// TIA Portal V16 export
// export: Created 2022-02-11T14:53:34.4841249Z, ExportSetting WithDefaults, DisplayName Totally Integrated Automation Portal, DisplayVersion V16 Update 1, DisplayName TIA Portal Version Control Interface, DisplayVersion V16, DisplayName TIA Portal Openness, DisplayVersion V16, DisplayName SINAMICS Startdrive Advanced, DisplayVersion V16 Update 5, DisplayName SINAMICS Startdrive G130, G150, S120, S150, SINAMICS MV, S210, DisplayVersion V16 Update 5, DisplayName SINAMICS Startdrive G110M, G120, G120C, G120D, G120P, G115D, DisplayVersion V16 Update 5, DisplayName STEP 7 Professional, DisplayVersion V16, DisplayName STEP 7 Safety, DisplayVersion V16, DisplayName WinCC Advanced, DisplayVersion V16, DisplayName SIMATIC Visualization Architect, DisplayVersion V16
FUNCTION_BLOCK "Сортировка"   // FB9, LAD
VERSION : 0.1
// Логика работы ПФМ
// stored: AutoNumber true, IsIECCheckEnabled false, UDAEnableTagReadback false
   VAR_INPUT
      packet_released : Bool;
   END_VAR
   VAR DB_SPECIFIC
      "TrigE76.4" : Bool;
      Trig_Dovod : Bool;
      LiftPushingPacket : Bool;
      TrigAutoPFM : Bool;
      Trig_Vill : Bool;
      Trig_Vill2 : Bool;
      LiftDownTrig : Bool;
      HaveSxema : Bool;
      NewPacket : Bool;
      LiftDown_old : Bool;
      LiftPushing_old : Bool;
      ForksForcingFinish : Bool;
      LiftForcingFinish : Bool;
      CommonForcingPacket : Bool;
      ElevatorLowering : Bool;
      NoGasketMode : Bool;   // режим без прокладки
      RampIsOn : Bool;
      RampIsOff : Bool;
      power_Vill : Bool := true;
      MakedLayer : Bool;
      AlarmLowerElevator : Bool;
      AlarmNotReadedPack : Bool;
      lift_return_trig : Bool;
      ramp_sync_old : Bool;
      BoardInLayerCounter : Int;
      LayersCounter : Int;
   END_VAR
   VAR
      Vibrator_KeyFazer { S7_SetPoint := 'True'} : "Vibrator";
      Run323_timer { S7_SetPoint := 'True'} : TP;
      LayerCounter { S7_SetPoint := 'True'} : "Adder";
   END_VAR
   VAR_TEMP
      Sert : Word;
   END_VAR
   VAR_TEMP   // added for the SCL form of the ladder/FBD networks
      _w1 : Bool;
      _w2 : Bool;
      _s5time1 : S5Time;
      _w3 : Bool;
      _w4 : Bool;
      _w5 : Bool;
      _s5time2 : S5Time;
   END_VAR
BEGIN

REGION Network 1: 221 группа на 14 моторов общий сигнал готовности
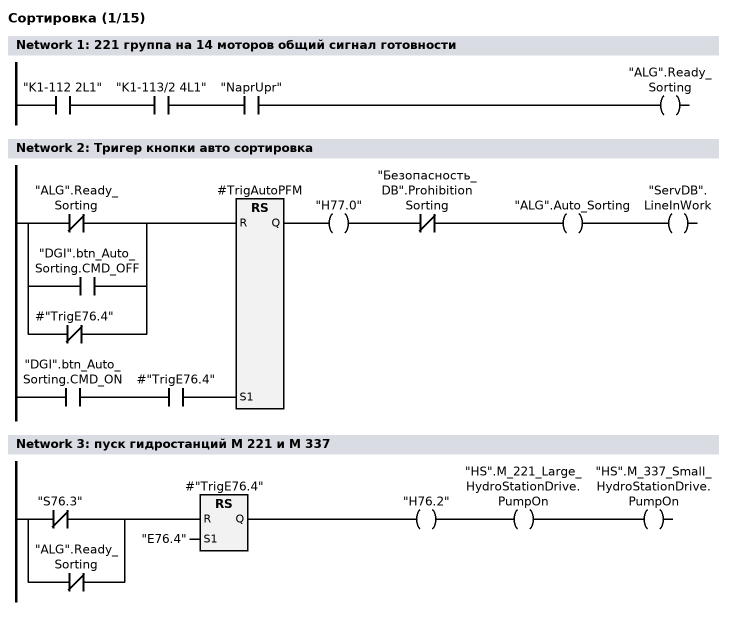
   RUNG wire#powerrail
      Contact( "K1-112 2L1" )
      Contact( "K1-113/2 4L1" )
      Contact( "NaprUpr" )
      Coil( "ALG".Ready_Sorting )
   END_RUNG
   // the same network as SCL:
   "ALG".Ready_Sorting := "K1-112 2L1" AND "K1-113/2 4L1" AND "NaprUpr";
END_REGION

REGION Network 2: Тригер кнопки авто сортировка
   RUNG wire#powerrail
      I_Contact( "ALG".Ready_Sorting )
      wire#w1
      S_RS(operand := #TrigAutoPFM, s1 := wire#w2)
      Coil( "H77.0" )
      I_Contact( "Безопасность_DB".ProhibitionSorting )
      Coil( "ALG".Auto_Sorting )
      Coil( "ServDB".LineInWork )
   END_RUNG
   RUNG wire#powerrail
      Contact( "DGI".btn_Auto_Sorting.CMD_OFF )
   END_RUNG wire#w1
   RUNG wire#powerrail
      I_Contact( #"TrigE76.4" )
   END_RUNG wire#w1
   RUNG wire#powerrail
      Contact( "DGI".btn_Auto_Sorting.CMD_ON )
      Contact( #"TrigE76.4" )
   END_RUNG wire#w2
   // the same network as SCL:
   IF NOT "ALG".Ready_Sorting OR "DGI".btn_Auto_Sorting.CMD_OFF OR NOT #"TrigE76.4" THEN
       #TrigAutoPFM := FALSE;   // RS flip-flop
   END_IF;
   IF "DGI".btn_Auto_Sorting.CMD_ON AND #"TrigE76.4" THEN #TrigAutoPFM := TRUE; END_IF;
   "H77.0" := #TrigAutoPFM;
   "ALG".Auto_Sorting := #TrigAutoPFM AND NOT "Безопасность_DB".ProhibitionSorting;
   "ServDB".LineInWork := "ALG".Auto_Sorting;
END_REGION

REGION Network 3: пуск гидростанций М 221 и M 337
   RUNG wire#powerrail
      I_Contact( "S76.3" )
      wire#w1
      S_RS(operand := #"TrigE76.4", s1 := "E76.4")
      Coil( "H76.2" )
      Coil( "HS".M_221_Large_HydroStationDrive.PumpOn )
      Coil( "HS".M_337_Small_HydroStationDrive.PumpOn )
   END_RUNG
   RUNG wire#powerrail
      I_Contact( "ALG".Ready_Sorting )
   END_RUNG wire#w1
   // the same network as SCL:
   IF NOT "S76.3" OR NOT "ALG".Ready_Sorting THEN
       #"TrigE76.4" := FALSE;   // RS flip-flop
   END_IF;
   IF "E76.4" THEN #"TrigE76.4" := TRUE; END_IF;
   "H76.2" := #"TrigE76.4";
   "HS".M_221_Large_HydroStationDrive.PumpOn := #"TrigE76.4";
   "HS".M_337_Small_HydroStationDrive.PumpOn := #"TrigE76.4";
END_REGION

REGION Network 4: Генерация аварии
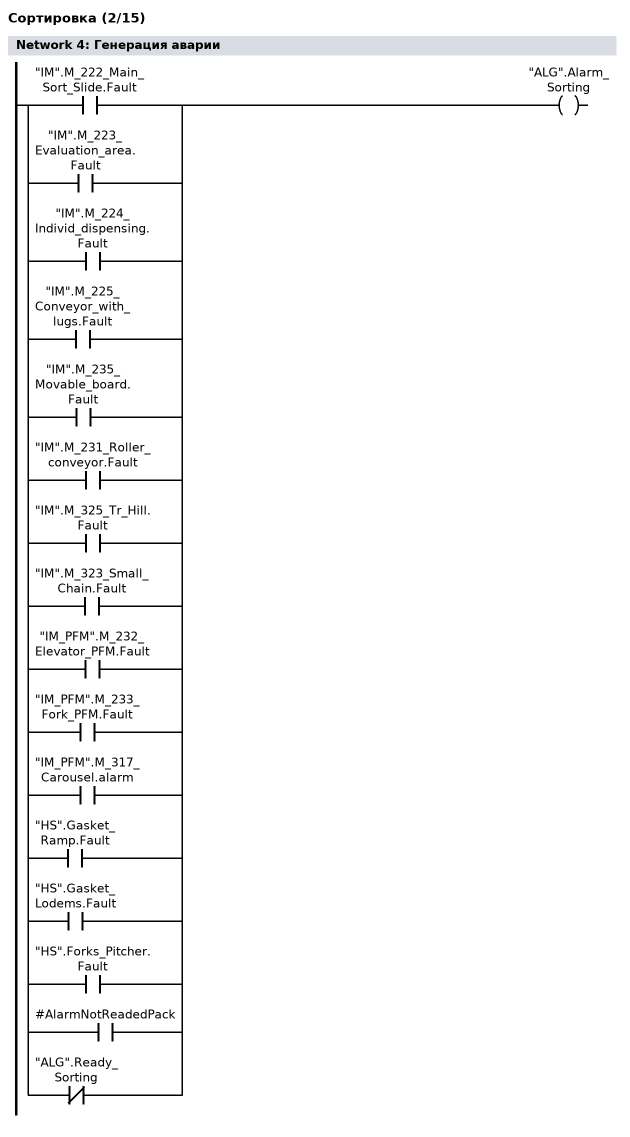
   RUNG wire#powerrail
      Contact( "IM".M_222_Main_Sort_Slide.Fault )
      wire#w1
      Coil( "ALG".Alarm_Sorting )
   END_RUNG
   RUNG wire#powerrail
      Contact( "IM".M_223_Evaluation_area.Fault )
   END_RUNG wire#w1
   RUNG wire#powerrail
      Contact( "IM".M_224_Individ_dispensing.Fault )
   END_RUNG wire#w1
   RUNG wire#powerrail
      Contact( "IM".M_225_Conveyor_with_lugs.Fault )
   END_RUNG wire#w1
   RUNG wire#powerrail
      Contact( "IM".M_235_Movable_board.Fault )
   END_RUNG wire#w1
   RUNG wire#powerrail
      Contact( "IM".M_231_Roller_conveyor.Fault )
   END_RUNG wire#w1
   RUNG wire#powerrail
      Contact( "IM".M_325_Tr_Hill.Fault )
   END_RUNG wire#w1
   RUNG wire#powerrail
      Contact( "IM".M_323_Small_Chain.Fault )
   END_RUNG wire#w1
   RUNG wire#powerrail
      Contact( "IM_PFM".M_232_Elevator_PFM.Fault )
   END_RUNG wire#w1
   RUNG wire#powerrail
      Contact( "IM_PFM".M_233_Fork_PFM.Fault )
   END_RUNG wire#w1
   RUNG wire#powerrail
      Contact( "IM_PFM".M_317_Carousel.alarm )
   END_RUNG wire#w1
   RUNG wire#powerrail
      Contact( "HS".Gasket_Ramp.Fault )
   END_RUNG wire#w1
   RUNG wire#powerrail
      Contact( "HS".Gasket_Lodems.Fault )
   END_RUNG wire#w1
   RUNG wire#powerrail
      Contact( "HS".Forks_Pitcher.Fault )
   END_RUNG wire#w1
   RUNG wire#powerrail
      Contact( #AlarmNotReadedPack )
   END_RUNG wire#w1
   RUNG wire#powerrail
      I_Contact( "ALG".Ready_Sorting )
   END_RUNG wire#w1
   // the same network as SCL:
   "ALG".Alarm_Sorting := "IM".M_222_Main_Sort_Slide.Fault OR "IM".M_223_Evaluation_area.Fault OR "IM".M_224_Individ_dispensing.Fault OR "IM".M_225_Conveyor_with_lugs.Fault OR "IM".M_235_Movable_board.Fault OR "IM".M_231_Roller_conveyor.Fault OR "IM".M_325_Tr_Hill.Fault OR "IM".M_323_Small_Chain.Fault OR "IM_PFM".M_232_Elevator_PFM.Fault OR "IM_PFM".M_233_Fork_PFM.Fault OR "IM_PFM".M_317_Carousel.alarm OR "HS".Gasket_Ramp.Fault OR "HS".Gasket_Lodems.Fault OR "HS".Forks_Pitcher.Fault OR #AlarmNotReadedPack OR NOT "ALG".Ready_Sorting;
END_REGION

REGION Network 5: Сбор аварий с других узлов + аварии не генерирующие останов линии
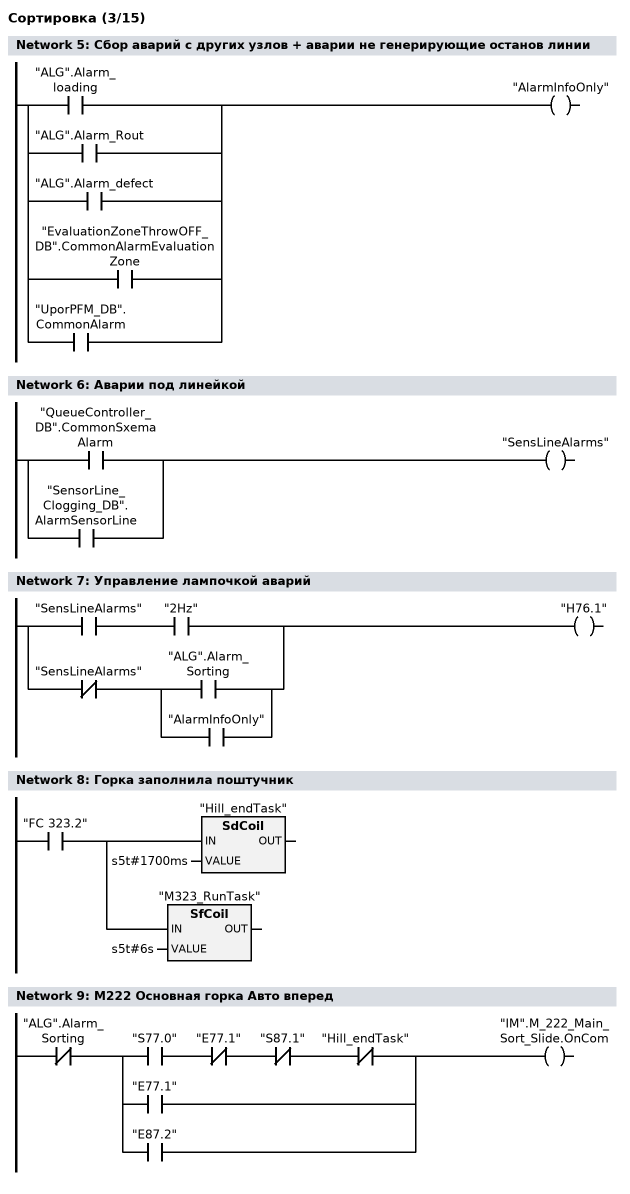
   RUNG wire#powerrail
      Contact( "ALG".Alarm_loading )
      wire#w1
      Coil( "AlarmInfoOnly" )
   END_RUNG
   RUNG wire#powerrail
      Contact( "ALG".Alarm_Rout )
   END_RUNG wire#w1
   RUNG wire#powerrail
      Contact( "ALG".Alarm_defect )
   END_RUNG wire#w1
   RUNG wire#powerrail
      Contact( "EvaluationZoneThrowOFF_DB".CommonAlarmEvaluationZone )
   END_RUNG wire#w1
   RUNG wire#powerrail
      Contact( "UporPFM_DB".CommonAlarm )
   END_RUNG wire#w1
   // the same network as SCL:
   "AlarmInfoOnly" := "ALG".Alarm_loading OR "ALG".Alarm_Rout OR "ALG".Alarm_defect OR "EvaluationZoneThrowOFF_DB".CommonAlarmEvaluationZone OR "UporPFM_DB".CommonAlarm;
END_REGION

REGION Network 6: Аварии под линейкой
   RUNG wire#powerrail
      Contact( "QueueController_DB".CommonSxemaAlarm )
      wire#w1
      Coil( "SensLineAlarms" )
   END_RUNG
   RUNG wire#powerrail
      Contact( "SensorLine_Clogging_DB".AlarmSensorLine )
   END_RUNG wire#w1
   // the same network as SCL:
   "SensLineAlarms" := "QueueController_DB".CommonSxemaAlarm OR "SensorLine_Clogging_DB".AlarmSensorLine;
END_REGION

REGION Network 7: Управление лампочкой аварий
   RUNG wire#powerrail
      Contact( "SensLineAlarms" )
      Contact( "2Hz" )
      wire#w1
      Coil( "H76.1" )
   END_RUNG
   RUNG wire#powerrail
      I_Contact( "SensLineAlarms" )
      wire#w2
      Contact( "ALG".Alarm_Sorting )
   END_RUNG wire#w1
   RUNG wire#w2
      Contact( "AlarmInfoOnly" )
   END_RUNG wire#w1
   // the same network as SCL:
   "H76.1" := ("SensLineAlarms" AND "2Hz") OR (NOT "SensLineAlarms" AND ("ALG".Alarm_Sorting OR "AlarmInfoOnly"));
END_REGION

REGION Network 8: Горка заполнила поштучник
   // no SCL statement known for SdCoil, SfCoil: written as a call
   #_w1 := "FC 323.2";
   SdCoil(in := "FC 323.2", value := s5t#1700ms, operand := "Hill_endTask");
   SfCoil(in := #_w1, value := s5t#6s, operand := "M323_RunTask");
END_REGION

REGION Network 9: М222 Основная горка Авто вперед
   RUNG wire#powerrail
      I_Contact( "ALG".Alarm_Sorting )
      wire#w1
      Contact( "S77.0" )
      I_Contact( "E77.1" )
      I_Contact( "S87.1" )
      I_Contact( "Hill_endTask" )
      wire#w2
      Coil( "IM".M_222_Main_Sort_Slide.OnCom )
   END_RUNG
   RUNG wire#w1
      Contact( "E77.1" )
   END_RUNG wire#w2
   RUNG wire#w1
      Contact( "E87.2" )
   END_RUNG wire#w2
   // the same network as SCL:
   "IM".M_222_Main_Sort_Slide.OnCom := NOT "ALG".Alarm_Sorting AND (("S77.0" AND NOT "E77.1" AND NOT "S87.1" AND NOT "Hill_endTask") OR "E77.1" OR "E87.2");
END_REGION

REGION Network 10: М222 Основная горка команда на движениее
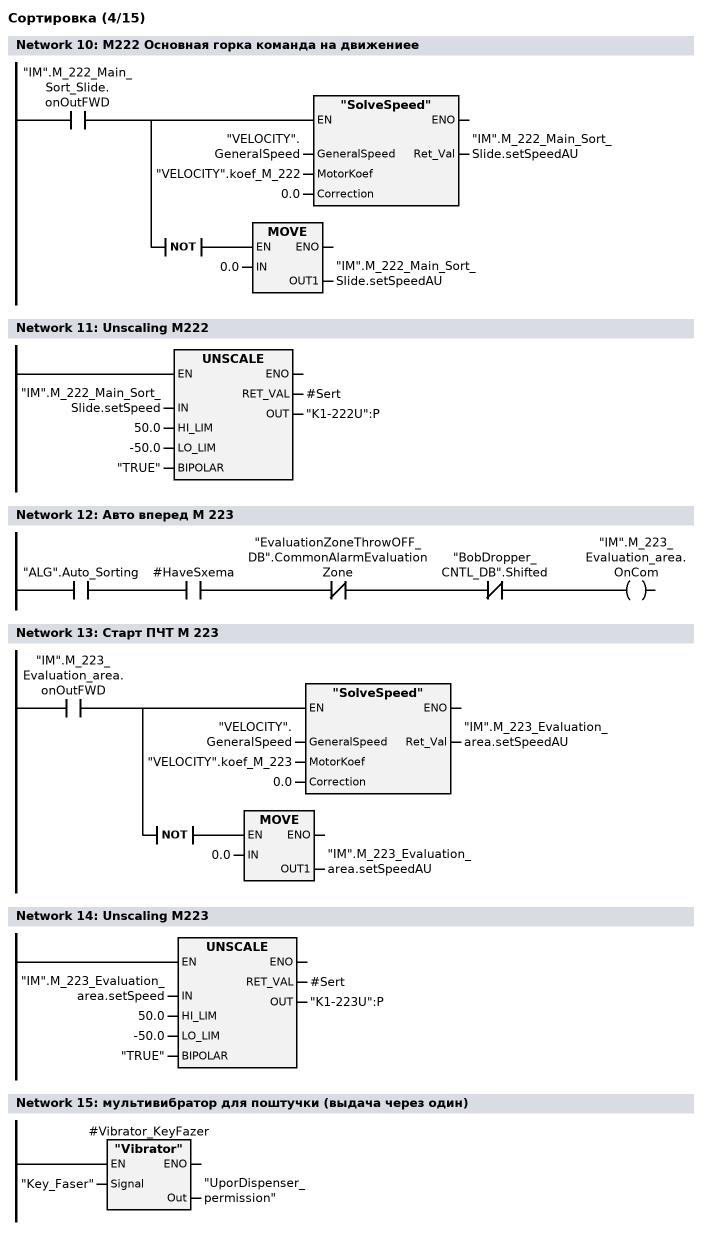
   RUNG wire#powerrail
      Contact( "IM".M_222_Main_Sort_Slide.onOutFWD )
      wire#w1
      "SolveSpeed"(GeneralSpeed := "VELOCITY".GeneralSpeed, MotorKoef := "VELOCITY".koef_M_222, Correction := 0.0, Ret_Val => "IM".M_222_Main_Sort_Slide.setSpeedAU)
   END_RUNG
   RUNG wire#w1
      Not()
      { S7_GenerateENO := "TRUE" } Move(in := 0.0, out1 => "IM".M_222_Main_Sort_Slide.setSpeedAU)
   END_RUNG
   // the same network as SCL:
   #_w1 := "IM".M_222_Main_Sort_Slide.onOutFWD;
   IF #_w1 THEN
       "IM".M_222_Main_Sort_Slide.setSpeedAU := "SolveSpeed"(GeneralSpeed := "VELOCITY".GeneralSpeed,
                               MotorKoef := "VELOCITY".koef_M_222,
                               Correction := 0.0);
   END_IF;
   IF NOT #_w1 THEN "IM".M_222_Main_Sort_Slide.setSpeedAU := 0.0; END_IF;
END_REGION

REGION Network 11: Unscaling M222
   RUNG wire#powerrail
      UNSCALE(IN := "IM".M_222_Main_Sort_Slide.setSpeed, HI_LIM := 50.0, LO_LIM := -50.0, BIPOLAR := "TRUE", RET_VAL => #Sert, OUT => "K1-222U":P)
   END_RUNG
   // the same network as SCL:
   #Sert := UNSCALE(IN := "IM".M_222_Main_Sort_Slide.setSpeed,
                    HI_LIM := 50.0,
                    LO_LIM := -50.0,
                    BIPOLAR := "TRUE",
                    OUT => "K1-222U":P);
END_REGION

REGION Network 12: Авто вперед M 223
   RUNG wire#powerrail
      Contact( "ALG".Auto_Sorting )
      Contact( #HaveSxema )
      I_Contact( "EvaluationZoneThrowOFF_DB".CommonAlarmEvaluationZone )
      I_Contact( "BobDropper_CNTL_DB".Shifted )
      Coil( "IM".M_223_Evaluation_area.OnCom )
   END_RUNG
   // the same network as SCL:
   "IM".M_223_Evaluation_area.OnCom := "ALG".Auto_Sorting AND #HaveSxema AND NOT "EvaluationZoneThrowOFF_DB".CommonAlarmEvaluationZone AND NOT "BobDropper_CNTL_DB".Shifted;
END_REGION

REGION Network 13: Старт ПЧТ М 223
   RUNG wire#powerrail
      Contact( "IM".M_223_Evaluation_area.onOutFWD )
      wire#w1
      "SolveSpeed"(GeneralSpeed := "VELOCITY".GeneralSpeed, MotorKoef := "VELOCITY".koef_M_223, Correction := 0.0, Ret_Val => "IM".M_223_Evaluation_area.setSpeedAU)
   END_RUNG
   RUNG wire#w1
      Not()
      { S7_GenerateENO := "TRUE" } Move(in := 0.0, out1 => "IM".M_223_Evaluation_area.setSpeedAU)
   END_RUNG
   // the same network as SCL:
   #_w1 := "IM".M_223_Evaluation_area.onOutFWD;
   IF #_w1 THEN
       "IM".M_223_Evaluation_area.setSpeedAU := "SolveSpeed"(GeneralSpeed := "VELOCITY".GeneralSpeed,
                               MotorKoef := "VELOCITY".koef_M_223,
                               Correction := 0.0);
   END_IF;
   IF NOT #_w1 THEN "IM".M_223_Evaluation_area.setSpeedAU := 0.0; END_IF;
END_REGION

REGION Network 14: Unscaling M223
   RUNG wire#powerrail
      UNSCALE(IN := "IM".M_223_Evaluation_area.setSpeed, HI_LIM := 50.0, LO_LIM := -50.0, BIPOLAR := "TRUE", RET_VAL => #Sert, OUT => "K1-223U":P)
   END_RUNG
   // the same network as SCL:
   #Sert := UNSCALE(IN := "IM".M_223_Evaluation_area.setSpeed,
                    HI_LIM := 50.0,
                    LO_LIM := -50.0,
                    BIPOLAR := "TRUE",
                    OUT => "K1-223U":P);
END_REGION

REGION Network 15: мультивибратор для поштучки (выдача через один)
   RUNG wire#powerrail
      #Vibrator_KeyFazer(Signal := "Key_Faser", Out => "UporDispenser_permission")
   END_RUNG
   // the same network as SCL:
   #Vibrator_KeyFazer(Signal := "Key_Faser", Out => "UporDispenser_permission");   // "Vibrator"
END_REGION

REGION Network 16: Есть схема для сортировки
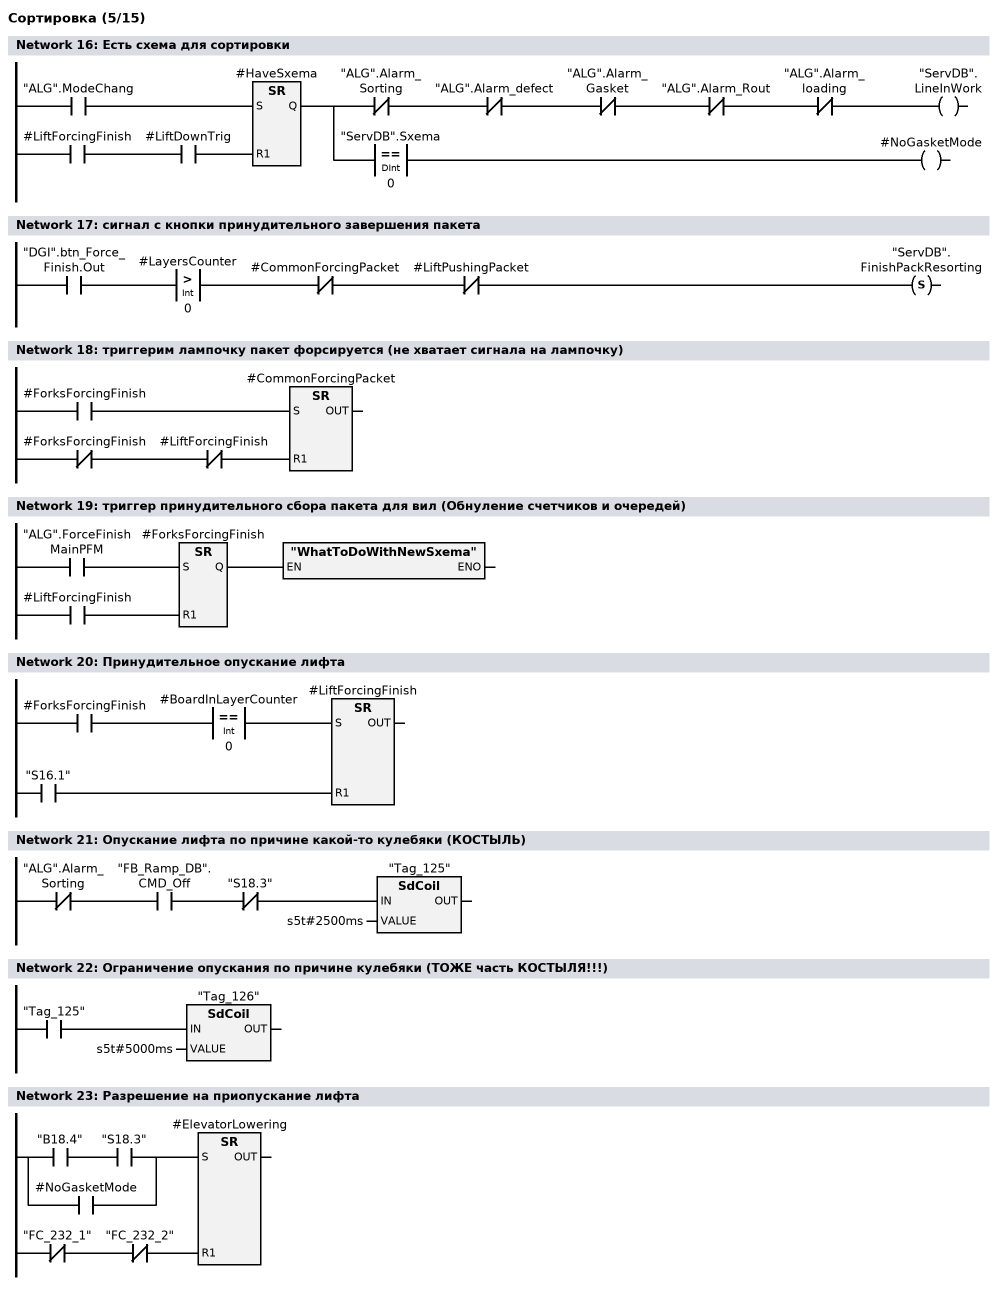
   RUNG wire#powerrail
      Contact( "ALG".ModeChang )
      S_SR(operand := #HaveSxema, r1 := wire#w1)
      wire#w2
      I_Contact( "ALG".Alarm_Sorting )
      I_Contact( "ALG".Alarm_defect )
      I_Contact( "ALG".Alarm_Gasket )
      I_Contact( "ALG".Alarm_Rout )
      I_Contact( "ALG".Alarm_loading )
      Coil( "ServDB".LineInWork )
   END_RUNG
   RUNG wire#powerrail
      Contact( #LiftForcingFinish )
      Contact( #LiftDownTrig )
   END_RUNG wire#w1
   RUNG wire#w2
      { S7_Templates := "SrcType := DInt" } EQ_Contact(in1 := "ServDB".Sxema, in2 := 0)
      Coil( #NoGasketMode )
   END_RUNG
   // the same network as SCL:
   IF "ALG".ModeChang THEN
       #HaveSxema := TRUE;   // SR flip-flop
   END_IF;
   IF #LiftForcingFinish AND #LiftDownTrig THEN #HaveSxema := FALSE; END_IF;
   "ServDB".LineInWork := #HaveSxema AND NOT "ALG".Alarm_Sorting AND NOT "ALG".Alarm_defect AND NOT "ALG".Alarm_Gasket AND NOT "ALG".Alarm_Rout AND NOT "ALG".Alarm_loading;
   #NoGasketMode := #HaveSxema AND ("ServDB".Sxema = 0);
END_REGION

REGION Network 17: сигнал с кнопки принудительного завершения пакета
   RUNG wire#powerrail
      Contact( "DGI".btn_Force_Finish.Out )
      { S7_Templates := "SrcType := Int" } GT_Contact(in1 := #LayersCounter, in2 := 0)
      I_Contact( #CommonForcingPacket )
      I_Contact( #LiftPushingPacket )
      S_Coil( "ServDB".FinishPackResorting )
   END_RUNG
   // the same network as SCL:
   IF "DGI".btn_Force_Finish.Out AND (#LayersCounter > 0) AND NOT #CommonForcingPacket AND NOT #LiftPushingPacket THEN
       "ServDB".FinishPackResorting := TRUE;
   END_IF;
END_REGION

REGION Network 18: триггерим лампочку пакет форсируется (не хватает сигнала на лампочку)
   RUNG wire#powerrail
      Contact( #ForksForcingFinish )
      S_SR(operand := #CommonForcingPacket, r1 := wire#w1)
   END_RUNG
   RUNG wire#powerrail
      I_Contact( #ForksForcingFinish )
      I_Contact( #LiftForcingFinish )
   END_RUNG wire#w1
   // the same network as SCL:
   IF #ForksForcingFinish THEN
       #CommonForcingPacket := TRUE;   // SR flip-flop
   END_IF;
   IF NOT #ForksForcingFinish AND NOT #LiftForcingFinish THEN #CommonForcingPacket := FALSE; END_IF;
END_REGION

REGION Network 19: триггер принудительного сбора пакета для вил (Обнуление счетчиков и очередей)
   RUNG wire#powerrail
      Contact( "ALG".ForceFinishMainPFM )
      S_SR(operand := #ForksForcingFinish, r1 := wire#w1)
      "WhatToDoWithNewSxema"()
   END_RUNG
   RUNG wire#powerrail
      Contact( #LiftForcingFinish )
   END_RUNG wire#w1
   // the same network as SCL:
   IF "ALG".ForceFinishMainPFM THEN
       #ForksForcingFinish := TRUE;   // SR flip-flop
   END_IF;
   IF #LiftForcingFinish THEN #ForksForcingFinish := FALSE; END_IF;
   IF #ForksForcingFinish THEN "WhatToDoWithNewSxema"(); END_IF;
END_REGION

REGION Network 20: Принудительное опускание лифта
   RUNG wire#powerrail
      Contact( #ForksForcingFinish )
      { S7_Templates := "SrcType := Int" } EQ_Contact(in1 := #BoardInLayerCounter, in2 := 0)
      S_SR(operand := #LiftForcingFinish, r1 := wire#w1)
   END_RUNG
   RUNG wire#powerrail
      Contact( "S16.1" )
   END_RUNG wire#w1
   // the same network as SCL:
   IF #ForksForcingFinish AND (#BoardInLayerCounter = 0) THEN
       #LiftForcingFinish := TRUE;   // SR flip-flop
   END_IF;
   IF "S16.1" THEN #LiftForcingFinish := FALSE; END_IF;
END_REGION

REGION Network 21: Опускание лифта по причине какой-то кулебяки (КОСТЫЛЬ)
   // no SCL statement known for SdCoil: written as a call
   SdCoil(in := NOT "ALG".Alarm_Sorting AND "FB_Ramp_DB".CMD_Off AND NOT "S18.3",
          value := s5t#2500ms,
          operand := "Tag_125");
END_REGION

REGION Network 22: Ограничение опускания по причине кулебяки (ТОЖЕ часть КОСТЫЛЯ!!!)
   // no SCL statement known for SdCoil: written as a call
   SdCoil(in := "Tag_125", value := s5t#5000ms, operand := "Tag_126");
END_REGION

REGION Network 23: Разрешение на приопускание лифта
   RUNG wire#powerrail
      Contact( "B18.4" )
      Contact( "S18.3" )
      wire#w1
      S_SR(operand := #ElevatorLowering, r1 := wire#w2)
   END_RUNG
   RUNG wire#powerrail
      Contact( #NoGasketMode )
   END_RUNG wire#w1
   RUNG wire#powerrail
      I_Contact( "FC_232_1" )
      I_Contact( "FC_232_2" )
   END_RUNG wire#w2
   // the same network as SCL:
   IF ("B18.4" AND "S18.3") OR #NoGasketMode THEN
       #ElevatorLowering := TRUE;   // SR flip-flop
   END_IF;
   IF NOT "FC_232_1" AND NOT "FC_232_2" THEN #ElevatorLowering := FALSE; END_IF;
END_REGION

REGION Network 24: Счёт слоёв
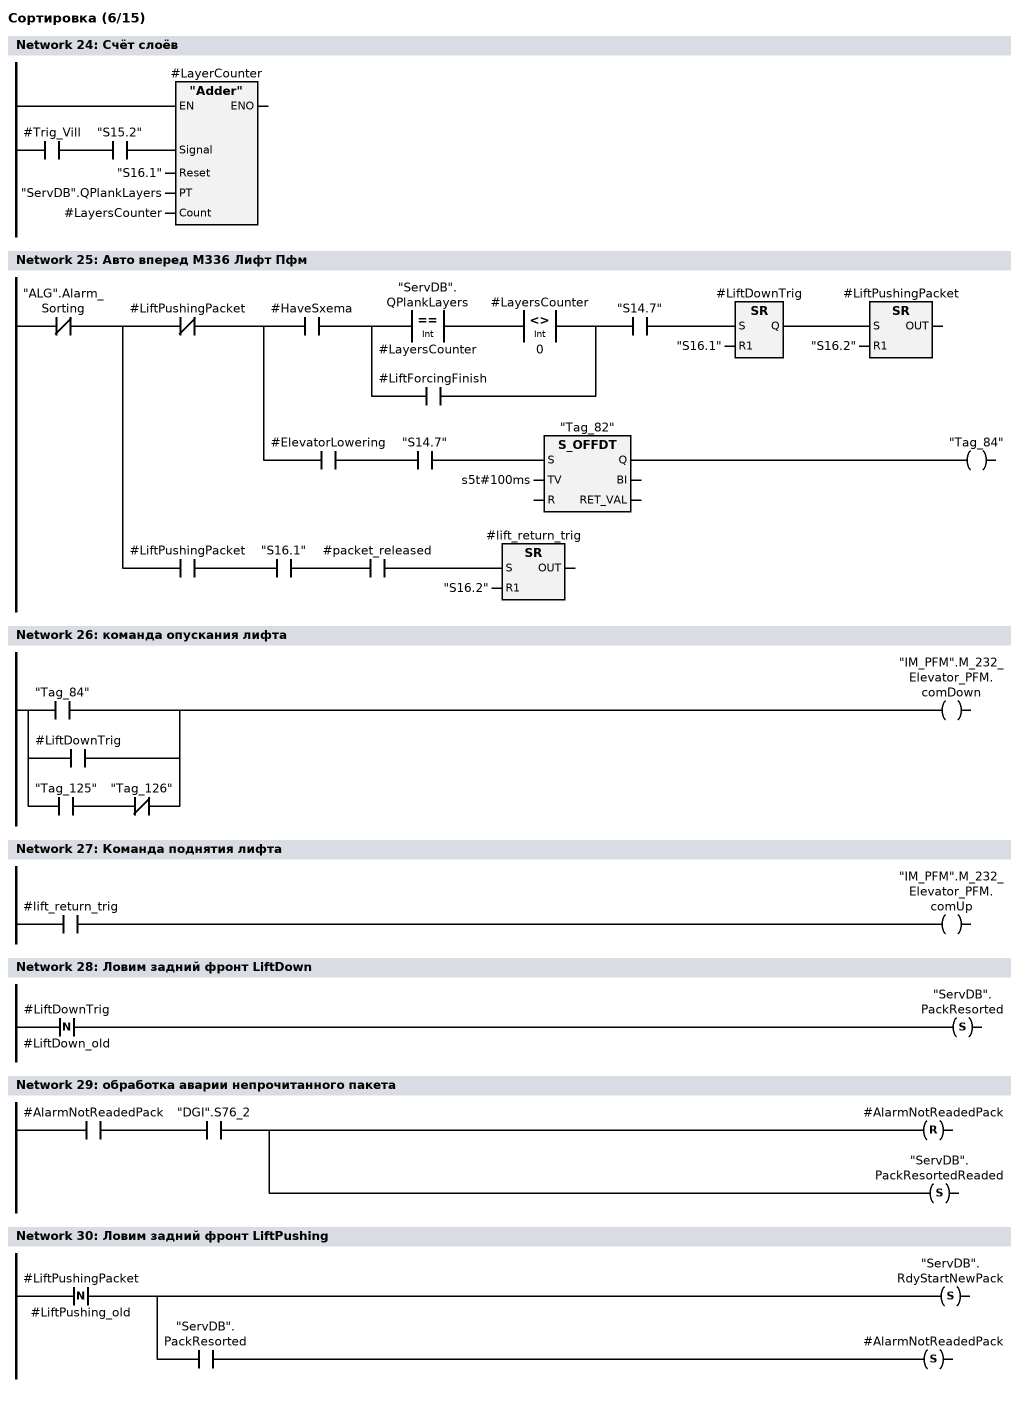
   RUNG wire#powerrail
      #LayerCounter(Signal := wire#w1, Reset := "S16.1", PT := "ServDB".QPlankLayers, Count := #LayersCounter)
   END_RUNG
   RUNG wire#powerrail
      Contact( #Trig_Vill )
      Contact( "S15.2" )
   END_RUNG wire#w1
   // the same network as SCL:
   #LayerCounter(Signal := #Trig_Vill AND "S15.2",   // "Adder"
                 Reset := "S16.1",
                 PT := "ServDB".QPlankLayers,
                 Count := #LayersCounter);
END_REGION

REGION Network 25: Авто вперед М336 Лифт Пфм
   RUNG wire#powerrail
      I_Contact( "ALG".Alarm_Sorting )
      wire#w1
      I_Contact( #LiftPushingPacket )
      wire#w2
      Contact( #HaveSxema )
      wire#w3
      { S7_Templates := "SrcType := Int" } EQ_Contact(in1 := "ServDB".QPlankLayers, in2 := #LayersCounter)
      { S7_Templates := "SrcType := Int" } NE_Contact(in1 := #LayersCounter, in2 := 0)
      wire#w4
      Contact( "S14.7" )
      S_SR(operand := #LiftDownTrig, r1 := "S16.1")
      S_SR(operand := #LiftPushingPacket, r1 := "S16.2")
   END_RUNG
   RUNG wire#w3
      Contact( #LiftForcingFinish )
   END_RUNG wire#w4
   RUNG wire#w2
      Contact( #ElevatorLowering )
      Contact( "S14.7" )
      S_OFFDT(T_NO := "Tag_82", TV := s5t#100ms, R :=, BI =>, RET_VAL =>)
      Coil( "Tag_84" )
   END_RUNG
   RUNG wire#w1
      Contact( #LiftPushingPacket )
      Contact( "S16.1" )
      Contact( #packet_released )
      S_SR(operand := #lift_return_trig, r1 := "S16.2")
   END_RUNG
   // the same network as SCL:
   #_w1 := NOT "ALG".Alarm_Sorting AND NOT #LiftPushingPacket;
   IF #_w1 AND #HaveSxema AND ((("ServDB".QPlankLayers = #LayersCounter) AND (#LayersCounter <> 0)) OR #LiftForcingFinish) AND "S14.7" THEN
       #LiftDownTrig := TRUE;   // SR flip-flop
   END_IF;
   IF "S16.1" THEN #LiftDownTrig := FALSE; END_IF;
   IF #LiftDownTrig THEN
       #LiftPushingPacket := TRUE;   // SR flip-flop
   END_IF;
   IF "S16.2" THEN #LiftPushingPacket := FALSE; END_IF;
   #_s5time1 := S_OFFDT(T_NO := "Tag_82",
                        S := #_w1 AND #ElevatorLowering AND "S14.7",
                        TV := s5t#100ms,
                        Q => #_w2);
   "Tag_84" := #_w2;
   IF NOT "ALG".Alarm_Sorting AND #LiftPushingPacket AND "S16.1" AND #packet_released THEN
       #lift_return_trig := TRUE;   // SR flip-flop
   END_IF;
   IF "S16.2" THEN #lift_return_trig := FALSE; END_IF;
END_REGION

REGION Network 26: команда опускания лифта
   RUNG wire#powerrail
      Contact( "Tag_84" )
      wire#w1
      Coil( "IM_PFM".M_232_Elevator_PFM.comDown )
   END_RUNG
   RUNG wire#powerrail
      Contact( #LiftDownTrig )
   END_RUNG wire#w1
   RUNG wire#powerrail
      Contact( "Tag_125" )
      I_Contact( "Tag_126" )
   END_RUNG wire#w1
   // the same network as SCL:
   "IM_PFM".M_232_Elevator_PFM.comDown := "Tag_84" OR #LiftDownTrig OR ("Tag_125" AND NOT "Tag_126");
END_REGION

REGION Network 27: Команда поднятия лифта
   RUNG wire#powerrail
      Contact( #lift_return_trig )
      Coil( "IM_PFM".M_232_Elevator_PFM.comUp )
   END_RUNG
   // the same network as SCL:
   "IM_PFM".M_232_Elevator_PFM.comUp := #lift_return_trig;
END_REGION

REGION Network 28: Ловим задний фронт LiftDown
   RUNG wire#powerrail
      N_Contact(operand := #LiftDownTrig, bit := #LiftDown_old)
      S_Coil( "ServDB".PackResorted )
   END_RUNG
   // the same network as SCL:
   #_w1 := NOT #LiftDownTrig AND #LiftDown_old;   // falling edge of #LiftDownTrig
   #LiftDown_old := #LiftDownTrig;
   IF #_w1 THEN "ServDB".PackResorted := TRUE; END_IF;
END_REGION

REGION Network 29: обработка аварии непрочитанного пакета
   RUNG wire#powerrail
      Contact( #AlarmNotReadedPack )
      Contact( "DGI".S76_2 )
      wire#w1
      R_Coil( #AlarmNotReadedPack )
   END_RUNG
   RUNG wire#w1
      S_Coil( "ServDB".PackResortedReaded )
   END_RUNG
   // the same network as SCL:
   #_w1 := #AlarmNotReadedPack AND "DGI".S76_2;
   IF #_w1 THEN
       #AlarmNotReadedPack := FALSE;
       "ServDB".PackResortedReaded := TRUE;
   END_IF;
END_REGION

REGION Network 30: Ловим задний фронт LiftPushing
   RUNG wire#powerrail
      N_Contact(operand := #LiftPushingPacket, bit := #LiftPushing_old)
      wire#w1
      S_Coil( "ServDB".RdyStartNewPack )
   END_RUNG
   RUNG wire#w1
      Contact( "ServDB".PackResorted )
      S_Coil( #AlarmNotReadedPack )
   END_RUNG
   // the same network as SCL:
   #_w1 := NOT #LiftPushingPacket AND #LiftPushing_old;   // falling edge of #LiftPushingPacket
   #LiftPushing_old := #LiftPushingPacket;
   IF #_w1 THEN "ServDB".RdyStartNewPack := TRUE; END_IF;
   IF #_w1 AND "ServDB".PackResorted THEN #AlarmNotReadedPack := TRUE; END_IF;
END_REGION

REGION Network 31: старт ПЧТ М232 лифт пфм ( TODO добавить контроль скорости)
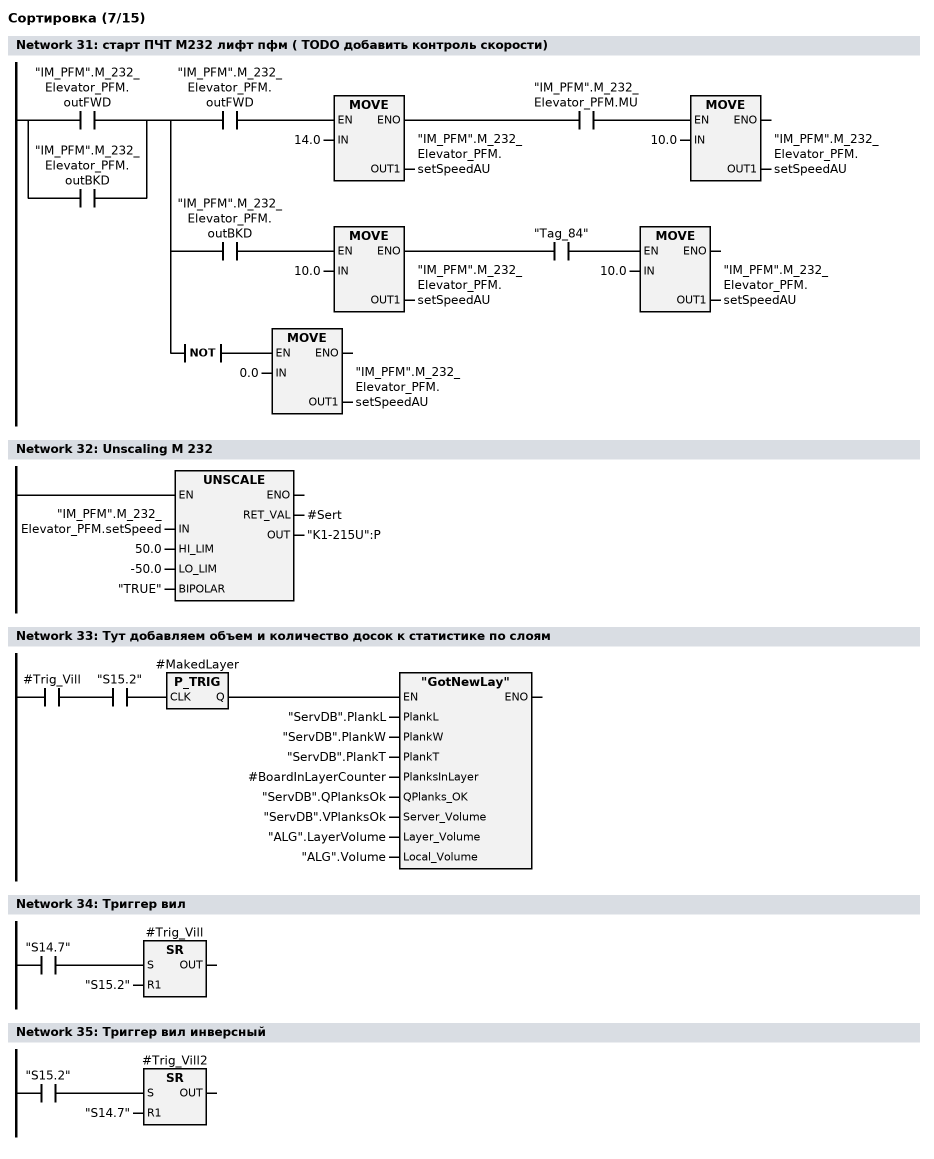
   RUNG wire#powerrail
      Contact( "IM_PFM".M_232_Elevator_PFM.outFWD )
      wire#w1
      Contact( "IM_PFM".M_232_Elevator_PFM.outFWD )
      { S7_GenerateENO := "TRUE" } Move(in := 14.0, out1 => "IM_PFM".M_232_Elevator_PFM.setSpeedAU)
      Contact( "IM_PFM".M_232_Elevator_PFM.MU )
      { S7_GenerateENO := "TRUE" } Move(in := 10.0, out1 => "IM_PFM".M_232_Elevator_PFM.setSpeedAU)
   END_RUNG
   RUNG wire#powerrail
      Contact( "IM_PFM".M_232_Elevator_PFM.outBKD )
   END_RUNG wire#w1
   RUNG wire#w1
      Contact( "IM_PFM".M_232_Elevator_PFM.outBKD )
      { S7_GenerateENO := "TRUE" } Move(in := 10.0, out1 => "IM_PFM".M_232_Elevator_PFM.setSpeedAU)
      Contact( "Tag_84" )
      { S7_GenerateENO := "TRUE" } Move(in := 10.0, out1 => "IM_PFM".M_232_Elevator_PFM.setSpeedAU)
   END_RUNG
   RUNG wire#w1
      Not()
      { S7_GenerateENO := "TRUE" } Move(in := 0.0, out1 => "IM_PFM".M_232_Elevator_PFM.setSpeedAU)
   END_RUNG
   // the same network as SCL:
   // ENO of a box is taken as its EN; it also drops when the box reports an error
   #_w1 := "IM_PFM".M_232_Elevator_PFM.outFWD OR "IM_PFM".M_232_Elevator_PFM.outBKD;
   #_w2 := #_w1 AND "IM_PFM".M_232_Elevator_PFM.outFWD;
   IF #_w2 THEN "IM_PFM".M_232_Elevator_PFM.setSpeedAU := 14.0; END_IF;
   IF #_w2 AND "IM_PFM".M_232_Elevator_PFM.MU THEN "IM_PFM".M_232_Elevator_PFM.setSpeedAU := 10.0; END_IF;
   #_w3 := #_w1 AND "IM_PFM".M_232_Elevator_PFM.outBKD;
   IF #_w3 THEN "IM_PFM".M_232_Elevator_PFM.setSpeedAU := 10.0; END_IF;
   IF #_w3 AND "Tag_84" THEN "IM_PFM".M_232_Elevator_PFM.setSpeedAU := 10.0; END_IF;
   IF NOT #_w1 THEN "IM_PFM".M_232_Elevator_PFM.setSpeedAU := 0.0; END_IF;
END_REGION

REGION Network 32: Unscaling M 232
   RUNG wire#powerrail
      UNSCALE(IN := "IM_PFM".M_232_Elevator_PFM.setSpeed, HI_LIM := 50.0, LO_LIM := -50.0, BIPOLAR := "TRUE", RET_VAL => #Sert, OUT => "K1-215U":P)
   END_RUNG
   // the same network as SCL:
   #Sert := UNSCALE(IN := "IM_PFM".M_232_Elevator_PFM.setSpeed,
                    HI_LIM := 50.0,
                    LO_LIM := -50.0,
                    BIPOLAR := "TRUE",
                    OUT => "K1-215U":P);
END_REGION

REGION Network 33: Тут добавляем объем и количество досок к статистике по слоям
   RUNG wire#powerrail
      Contact( #Trig_Vill )
      Contact( "S15.2" )
      P_Trig( #MakedLayer )
      "GotNewLay"(PlankL := "ServDB".PlankL, PlankW := "ServDB".PlankW, PlankT := "ServDB".PlankT, PlanksInLayer := #BoardInLayerCounter, QPlanks_OK := "ServDB".QPlanksOk, Server_Volume := "ServDB".VPlanksOk, Layer_Volume := "ALG".LayerVolume, Local_Volume := "ALG".Volume)
   END_RUNG
   // the same network as SCL:
   #_w1 := #Trig_Vill AND "S15.2";
   #_w2 := #_w1 AND NOT #MakedLayer;   // rising edge
   #MakedLayer := #_w1;
   IF #_w2 THEN
       "GotNewLay"(PlankL := "ServDB".PlankL,
                   PlankW := "ServDB".PlankW,
                   PlankT := "ServDB".PlankT,
                   PlanksInLayer := #BoardInLayerCounter,
                   QPlanks_OK := "ServDB".QPlanksOk,
                   Server_Volume := "ServDB".VPlanksOk,
                   Layer_Volume := "ALG".LayerVolume,
                   Local_Volume := "ALG".Volume);
   END_IF;
END_REGION

REGION Network 34: Триггер вил
   RUNG wire#powerrail
      Contact( "S14.7" )
      S_SR(operand := #Trig_Vill, r1 := "S15.2")
   END_RUNG
   // the same network as SCL:
   IF "S14.7" THEN
       #Trig_Vill := TRUE;   // SR flip-flop
   END_IF;
   IF "S15.2" THEN #Trig_Vill := FALSE; END_IF;
END_REGION

REGION Network 35: Триггер вил инверсный
   RUNG wire#powerrail
      Contact( "S15.2" )
      S_SR(operand := #Trig_Vill2, r1 := "S14.7")
   END_RUNG
   // the same network as SCL:
   IF "S15.2" THEN
       #Trig_Vill2 := TRUE;   // SR flip-flop
   END_IF;
   IF "S14.7" THEN #Trig_Vill2 := FALSE; END_IF;
END_REGION

REGION Network 36: Контроль кейфазеров на М225 и Счет досок на слой ПФМ (Счет не вызываем)
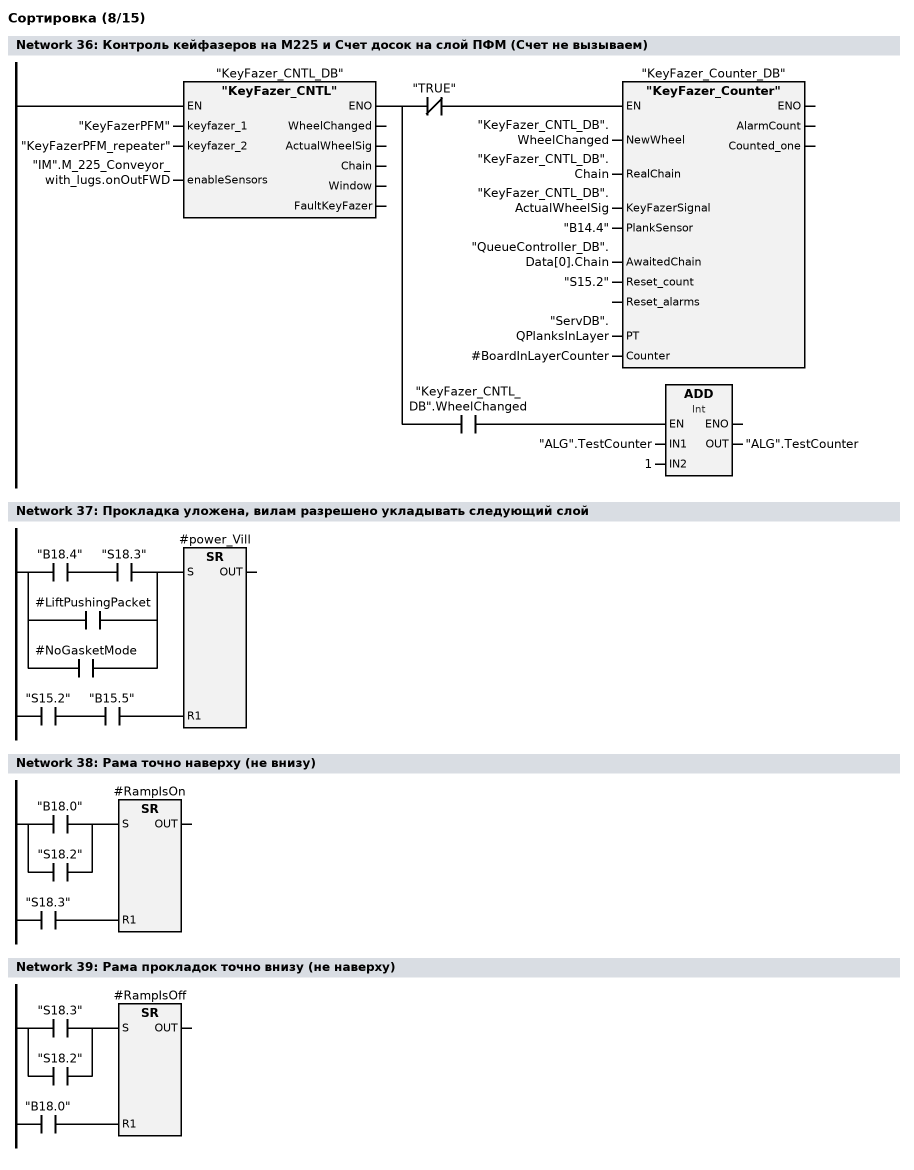
   RUNG wire#powerrail
      "KeyFazer_CNTL_DB"(keyfazer_1 := "KeyFazerPFM", keyfazer_2 := "KeyFazerPFM_repeater", enableSensors := "IM".M_225_Conveyor_with_lugs.onOutFWD, WheelChanged =>, ActualWheelSig =>, Chain =>, Window =>, FaultKeyFazer =>)
      wire#w1
      I_Contact( "TRUE" )
      "KeyFazer_Counter_DB"(NewWheel := "KeyFazer_CNTL_DB".WheelChanged, RealChain := "KeyFazer_CNTL_DB".Chain, KeyFazerSignal := "KeyFazer_CNTL_DB".ActualWheelSig, PlankSensor := "B14.4", AwaitedChain := "QueueController_DB".Data[0].Chain, Reset_count := "S15.2", Reset_alarms :=, PT := "ServDB".QPlanksInLayer, "Counter" := #BoardInLayerCounter, AlarmCount =>, Counted_one =>)
   END_RUNG
   RUNG wire#w1
      Contact( "KeyFazer_CNTL_DB".WheelChanged )
      { S7_Templates := "SrcType := Int"; S7_GenerateENO := "TRUE" } Add(in1 := "ALG".TestCounter, in2 := 1, out => "ALG".TestCounter)
   END_RUNG
   // the same network as SCL:
   "KeyFazer_CNTL_DB"(keyfazer_1 := "KeyFazerPFM",   // "KeyFazer_CNTL"
                      keyfazer_2 := "KeyFazerPFM_repeater",
                      enableSensors := "IM".M_225_Conveyor_with_lugs.onOutFWD,
                      ENO => #_w1);
   IF #_w1 AND NOT "TRUE" THEN
       "KeyFazer_Counter_DB"(NewWheel := "KeyFazer_CNTL_DB".WheelChanged,   // "KeyFazer_Counter"
                             RealChain := "KeyFazer_CNTL_DB".Chain,
                             KeyFazerSignal := "KeyFazer_CNTL_DB".ActualWheelSig,
                             PlankSensor := "B14.4",
                             AwaitedChain := "QueueController_DB".Data[0].Chain,
                             Reset_count := "S15.2",
                             PT := "ServDB".QPlanksInLayer,
                             "Counter" := #BoardInLayerCounter);
   END_IF;
   IF #_w1 AND "KeyFazer_CNTL_DB".WheelChanged THEN "ALG".TestCounter := "ALG".TestCounter + 1; END_IF;
END_REGION

REGION Network 37: Прокладка уложена, вилам разрешено укладывать следующий слой
   RUNG wire#powerrail
      Contact( "B18.4" )
      Contact( "S18.3" )
      wire#w1
      S_SR(operand := #power_Vill, r1 := wire#w2)
   END_RUNG
   RUNG wire#powerrail
      Contact( #LiftPushingPacket )
   END_RUNG wire#w1
   RUNG wire#powerrail
      Contact( #NoGasketMode )
   END_RUNG wire#w1
   RUNG wire#powerrail
      Contact( "S15.2" )
      Contact( "B15.5" )
   END_RUNG wire#w2
   // the same network as SCL:
   IF ("B18.4" AND "S18.3") OR #LiftPushingPacket OR #NoGasketMode THEN
       #power_Vill := TRUE;   // SR flip-flop
   END_IF;
   IF "S15.2" AND "B15.5" THEN #power_Vill := FALSE; END_IF;
END_REGION

REGION Network 38: Рама точно наверху (не внизу)
   RUNG wire#powerrail
      Contact( "B18.0" )
      wire#w1
      S_SR(operand := #RampIsOn, r1 := wire#w2)
   END_RUNG
   RUNG wire#powerrail
      Contact( "S18.2" )
   END_RUNG wire#w1
   RUNG wire#powerrail
      Contact( "S18.3" )
   END_RUNG wire#w2
   // the same network as SCL:
   IF "B18.0" OR "S18.2" THEN
       #RampIsOn := TRUE;   // SR flip-flop
   END_IF;
   IF "S18.3" THEN #RampIsOn := FALSE; END_IF;
END_REGION

REGION Network 39: Рама прокладок точно внизу (не наверху)
   RUNG wire#powerrail
      Contact( "S18.3" )
      wire#w1
      S_SR(operand := #RampIsOff, r1 := wire#w2)
   END_RUNG
   RUNG wire#powerrail
      Contact( "S18.2" )
   END_RUNG wire#w1
   RUNG wire#powerrail
      Contact( "B18.0" )
   END_RUNG wire#w2
   // the same network as SCL:
   IF "S18.3" OR "S18.2" THEN
       #RampIsOff := TRUE;   // SR flip-flop
   END_IF;
   IF "B18.0" THEN #RampIsOff := FALSE; END_IF;
END_REGION

REGION Network 40: M 233 вилы авто
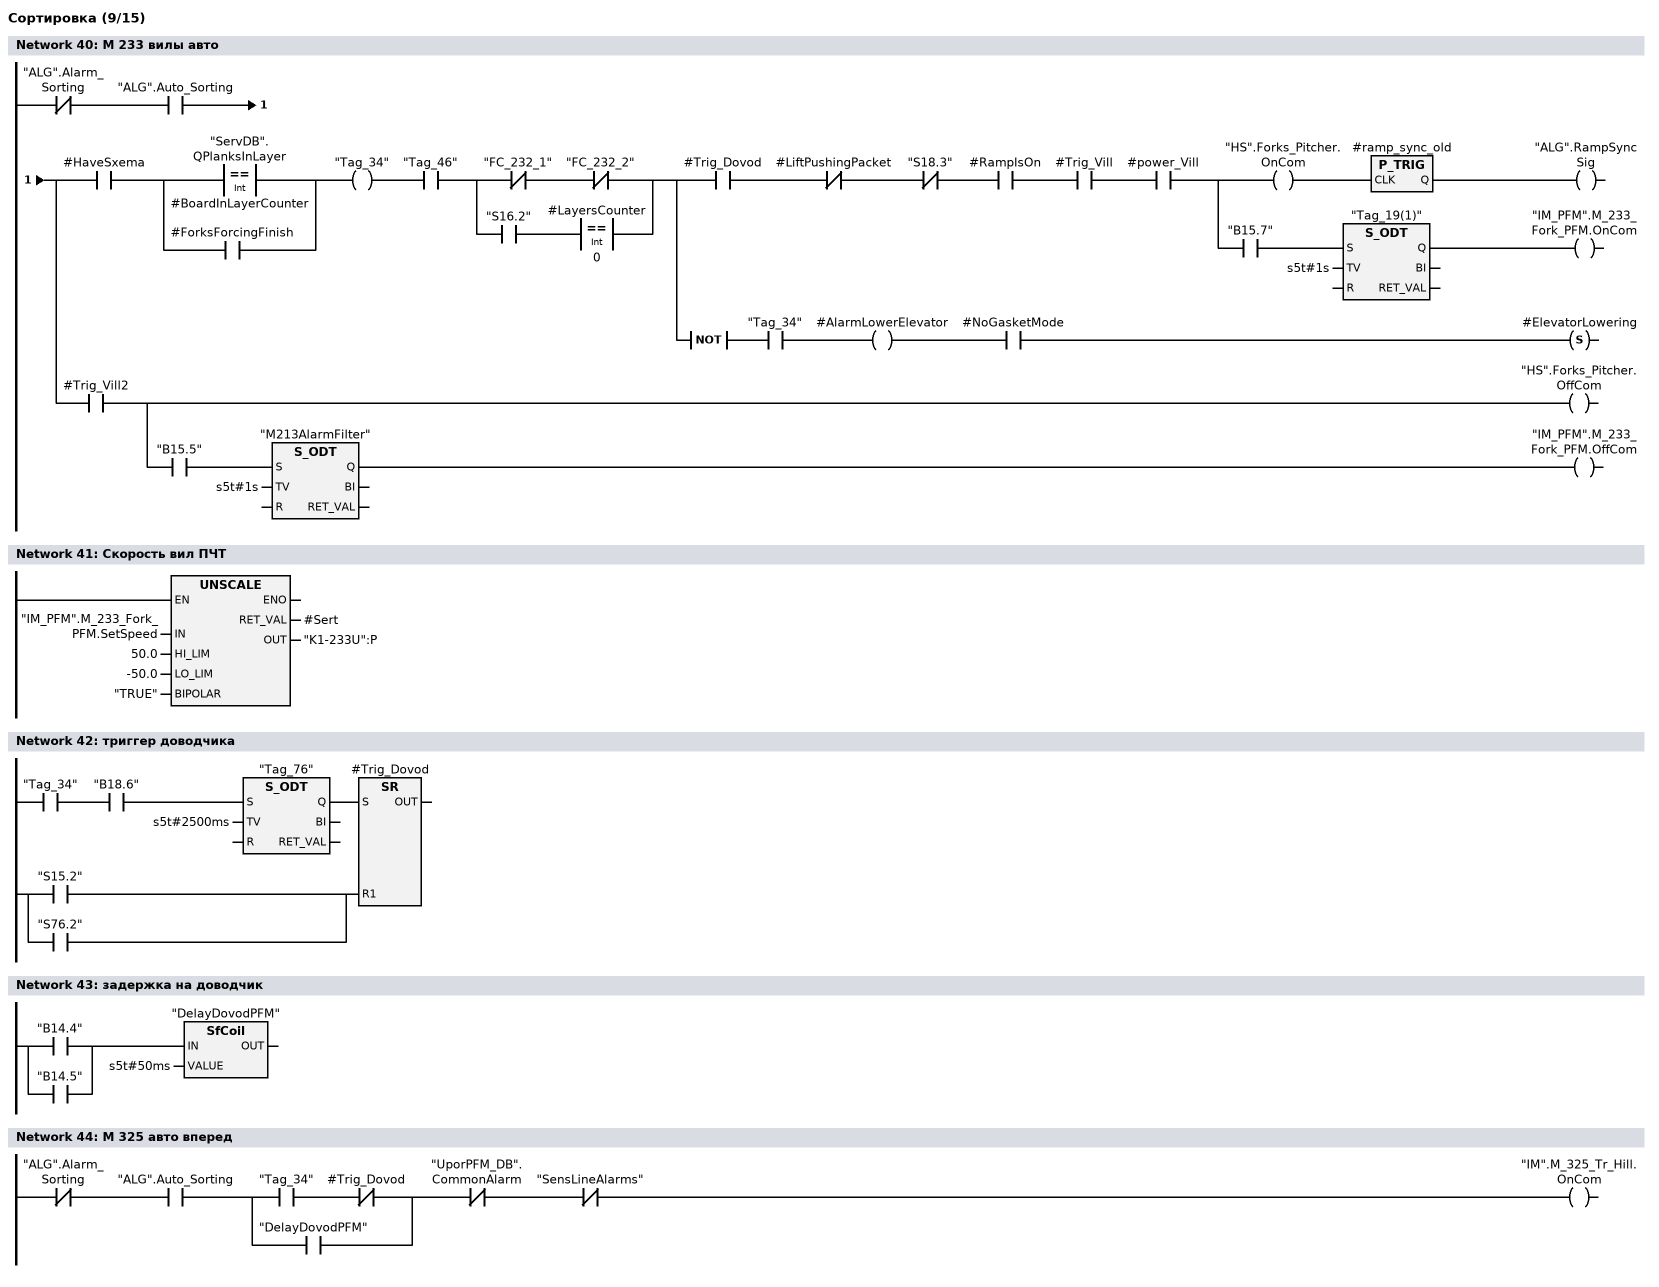
   RUNG wire#powerrail
      I_Contact( "ALG".Alarm_Sorting )
      Contact( "ALG".Auto_Sorting )
      wire#w1
      Contact( #HaveSxema )
      wire#w2
      { S7_Templates := "SrcType := Int" } EQ_Contact(in1 := "ServDB".QPlanksInLayer, in2 := #BoardInLayerCounter)
      wire#w3
      Coil( "Tag_34" )
      Contact( "Tag_46" )
      wire#w4
      I_Contact( "FC_232_1" )
      I_Contact( "FC_232_2" )
      wire#w5
      Contact( #Trig_Dovod )
      I_Contact( #LiftPushingPacket )
      I_Contact( "S18.3" )
      Contact( #RampIsOn )
      Contact( #Trig_Vill )
      Contact( #power_Vill )
      wire#w6
      Coil( "HS".Forks_Pitcher.OnCom )
      P_Trig( #ramp_sync_old )
      Coil( "ALG".RampSyncSig )
   END_RUNG
   RUNG wire#w2
      Contact( #ForksForcingFinish )
   END_RUNG wire#w3
   RUNG wire#w4
      Contact( "S16.2" )
      { S7_Templates := "SrcType := Int" } EQ_Contact(in1 := #LayersCounter, in2 := 0)
   END_RUNG wire#w5
   RUNG wire#w6
      Contact( "B15.7" )
      S_ODT(T_NO := "Tag_19(1)", TV := s5t#1s, R :=, BI =>, RET_VAL =>)
      Coil( "IM_PFM".M_233_Fork_PFM.OnCom )
   END_RUNG
   RUNG wire#w5
      Not()
      Contact( "Tag_34" )
      Coil( #AlarmLowerElevator )
      Contact( #NoGasketMode )
      S_Coil( #ElevatorLowering )
   END_RUNG
   RUNG wire#w1
      Contact( #Trig_Vill2 )
      wire#w7
      Coil( "HS".Forks_Pitcher.OffCom )
   END_RUNG
   RUNG wire#w7
      Contact( "B15.5" )
      S_ODT(T_NO := "M213AlarmFilter", TV := s5t#1s, R :=, BI =>, RET_VAL =>)
      Coil( "IM_PFM".M_233_Fork_PFM.OffCom )
   END_RUNG
   // the same network as SCL:
   #_w1 := NOT "ALG".Alarm_Sorting AND "ALG".Auto_Sorting;
   "Tag_34" := #_w1 AND #HaveSxema AND (("ServDB".QPlanksInLayer = #BoardInLayerCounter) OR #ForksForcingFinish);
   #_w2 := "Tag_34" AND "Tag_46" AND ((NOT "FC_232_1" AND NOT "FC_232_2") OR ("S16.2" AND (#LayersCounter = 0)));
   "HS".Forks_Pitcher.OnCom := #_w2 AND #Trig_Dovod AND NOT #LiftPushingPacket AND NOT "S18.3" AND #RampIsOn AND #Trig_Vill AND #power_Vill;
   #_w3 := "HS".Forks_Pitcher.OnCom AND NOT #ramp_sync_old;   // rising edge
   #ramp_sync_old := "HS".Forks_Pitcher.OnCom;
   "ALG".RampSyncSig := #_w3;
   #_s5time1 := S_ODT(T_NO := "Tag_19(1)", S := "HS".Forks_Pitcher.OnCom AND "B15.7", TV := s5t#1s, Q => #_w4);
   "IM_PFM".M_233_Fork_PFM.OnCom := #_w4;
   #AlarmLowerElevator := NOT #_w2 AND "Tag_34";
   IF #AlarmLowerElevator AND #NoGasketMode THEN #ElevatorLowering := TRUE; END_IF;
   "HS".Forks_Pitcher.OffCom := #_w1 AND #Trig_Vill2;
   #_s5time2 := S_ODT(T_NO := "M213AlarmFilter",
                      S := "HS".Forks_Pitcher.OffCom AND "B15.5",
                      TV := s5t#1s,
                      Q => #_w5);
   "IM_PFM".M_233_Fork_PFM.OffCom := #_w5;
END_REGION

REGION Network 41: Скорость вил ПЧТ
   RUNG wire#powerrail
      UNSCALE(IN := "IM_PFM".M_233_Fork_PFM.SetSpeed, HI_LIM := 50.0, LO_LIM := -50.0, BIPOLAR := "TRUE", RET_VAL => #Sert, OUT => "K1-233U":P)
   END_RUNG
   // the same network as SCL:
   #Sert := UNSCALE(IN := "IM_PFM".M_233_Fork_PFM.SetSpeed,
                    HI_LIM := 50.0,
                    LO_LIM := -50.0,
                    BIPOLAR := "TRUE",
                    OUT => "K1-233U":P);
END_REGION

REGION Network 42: триггер доводчика
   RUNG wire#powerrail
      Contact( "Tag_34" )
      Contact( "B18.6" )
      S_ODT(T_NO := "Tag_76", TV := s5t#2500ms, R :=, BI =>, RET_VAL =>)
      S_SR(operand := #Trig_Dovod, r1 := wire#w1)
   END_RUNG
   RUNG wire#powerrail
      Contact( "S15.2" )
   END_RUNG wire#w1
   RUNG wire#powerrail
      Contact( "S76.2" )
   END_RUNG wire#w1
   // the same network as SCL:
   #_s5time1 := S_ODT(T_NO := "Tag_76", S := "Tag_34" AND "B18.6", TV := s5t#2500ms, Q => #_w1);
   IF #_w1 THEN
       #Trig_Dovod := TRUE;   // SR flip-flop
   END_IF;
   IF "S15.2" OR "S76.2" THEN #Trig_Dovod := FALSE; END_IF;
END_REGION

REGION Network 43: задержка на доводчик
   // no SCL statement known for SfCoil: written as a call
   SfCoil(in := "B14.4" OR "B14.5", value := s5t#50ms, operand := "DelayDovodPFM");
END_REGION

REGION Network 44: M 325 авто вперед
   RUNG wire#powerrail
      I_Contact( "ALG".Alarm_Sorting )
      Contact( "ALG".Auto_Sorting )
      wire#w1
      Contact( "Tag_34" )
      I_Contact( #Trig_Dovod )
      wire#w2
      I_Contact( "UporPFM_DB".CommonAlarm )
      I_Contact( "SensLineAlarms" )
      Coil( "IM".M_325_Tr_Hill.OnCom )
   END_RUNG
   RUNG wire#w1
      Contact( "DelayDovodPFM" )
   END_RUNG wire#w2
   // the same network as SCL:
   "IM".M_325_Tr_Hill.OnCom := NOT "ALG".Alarm_Sorting AND "ALG".Auto_Sorting AND (("Tag_34" AND NOT #Trig_Dovod) OR "DelayDovodPFM") AND NOT "UporPFM_DB".CommonAlarm AND NOT "SensLineAlarms";
END_REGION

REGION Network 45: Старт ПЧТ 325
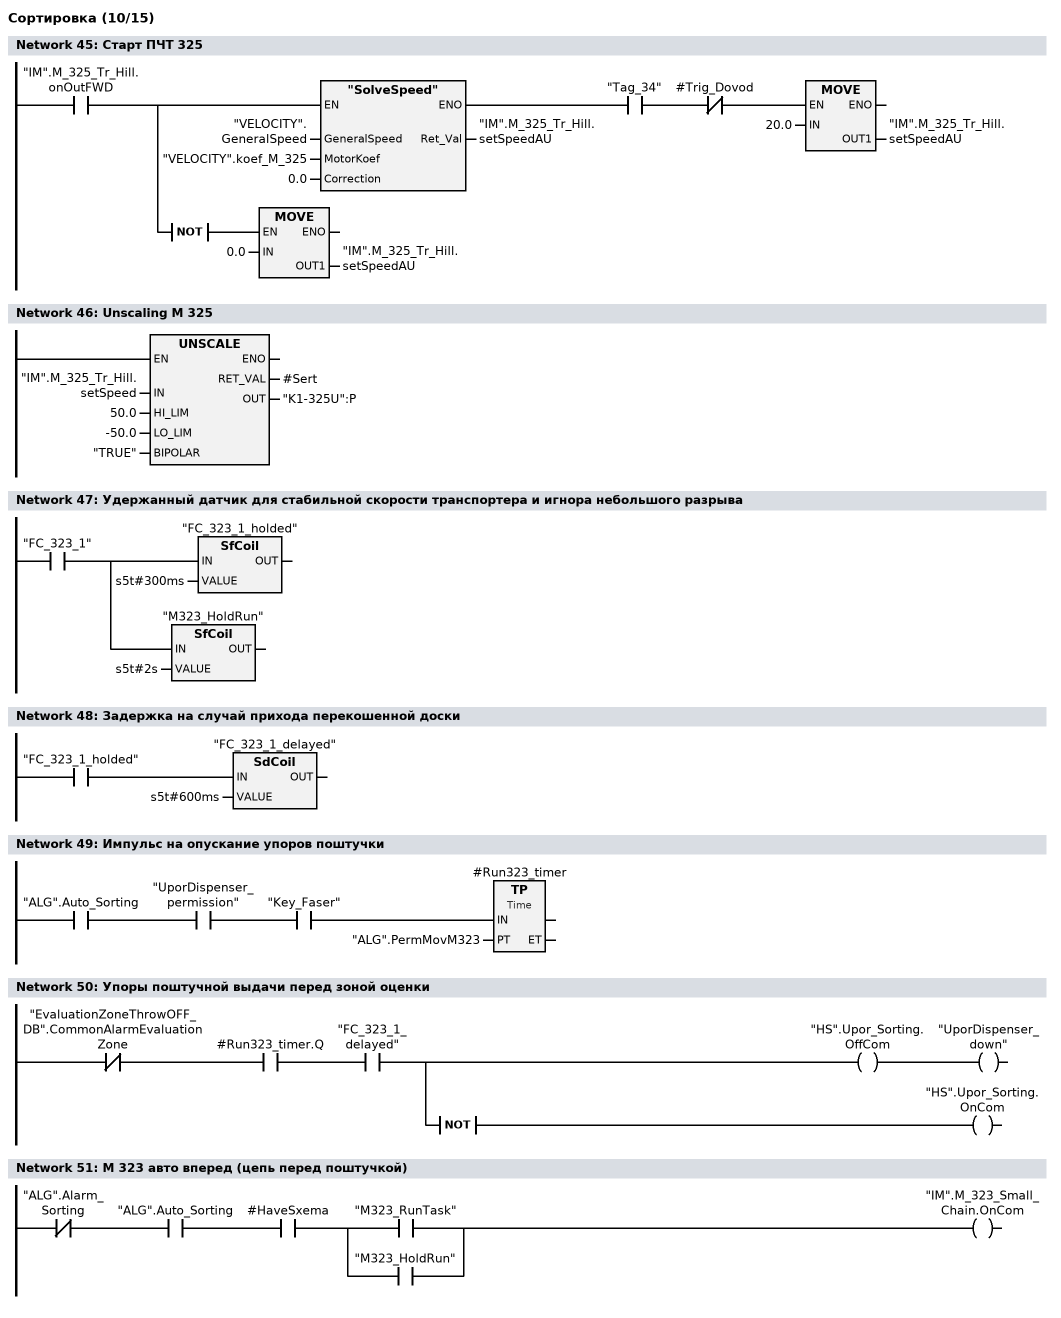
   RUNG wire#powerrail
      Contact( "IM".M_325_Tr_Hill.onOutFWD )
      wire#w1
      "SolveSpeed"(GeneralSpeed := "VELOCITY".GeneralSpeed, MotorKoef := "VELOCITY".koef_M_325, Correction := 0.0, Ret_Val => "IM".M_325_Tr_Hill.setSpeedAU)
      Contact( "Tag_34" )
      I_Contact( #Trig_Dovod )
      { S7_GenerateENO := "TRUE" } Move(in := 20.0, out1 => "IM".M_325_Tr_Hill.setSpeedAU)
   END_RUNG
   RUNG wire#w1
      Not()
      { S7_GenerateENO := "TRUE" } Move(in := 0.0, out1 => "IM".M_325_Tr_Hill.setSpeedAU)
   END_RUNG
   // the same network as SCL:
   #_w2 := "IM".M_325_Tr_Hill.onOutFWD;
   "IM".M_325_Tr_Hill.setSpeedAU := "SolveSpeed"(EN := "IM".M_325_Tr_Hill.onOutFWD,
                           GeneralSpeed := "VELOCITY".GeneralSpeed,
                           MotorKoef := "VELOCITY".koef_M_325,
                           Correction := 0.0,
                           ENO => #_w1);
   IF #_w1 AND "Tag_34" AND NOT #Trig_Dovod THEN "IM".M_325_Tr_Hill.setSpeedAU := 20.0; END_IF;
   IF NOT #_w2 THEN "IM".M_325_Tr_Hill.setSpeedAU := 0.0; END_IF;
END_REGION

REGION Network 46: Unscaling M 325
   RUNG wire#powerrail
      UNSCALE(IN := "IM".M_325_Tr_Hill.setSpeed, HI_LIM := 50.0, LO_LIM := -50.0, BIPOLAR := "TRUE", RET_VAL => #Sert, OUT => "K1-325U":P)
   END_RUNG
   // the same network as SCL:
   #Sert := UNSCALE(IN := "IM".M_325_Tr_Hill.setSpeed,
                    HI_LIM := 50.0,
                    LO_LIM := -50.0,
                    BIPOLAR := "TRUE",
                    OUT => "K1-325U":P);
END_REGION

REGION Network 47: Удержанный датчик для стабильной скорости транспортера и игнора небольшого разрыва
   // no SCL statement known for SfCoil: written as a call
   #_w1 := "FC_323_1";
   SfCoil(in := "FC_323_1", value := s5t#300ms, operand := "FC_323_1_holded");
   SfCoil(in := #_w1, value := s5t#2s, operand := "M323_HoldRun");
END_REGION

REGION Network 48: Задержка на случай прихода перекошенной доски
   // no SCL statement known for SdCoil: written as a call
   SdCoil(in := "FC_323_1_holded", value := s5t#600ms, operand := "FC_323_1_delayed");
END_REGION

REGION Network 49: Импульс на опускание упоров поштучки
   RUNG wire#powerrail
      Contact( "ALG".Auto_Sorting )
      Contact( "UporDispenser_permission" )
      Contact( "Key_Faser" )
      { S7_Templates := "time_type := Time" } #Run323_timer.TP(pt := "ALG".PermMovM323, et =>)
   END_RUNG
   // the same network as SCL:
   #Run323_timer.TP(IN := "ALG".Auto_Sorting AND "UporDispenser_permission" AND "Key_Faser",
                    PT := "ALG".PermMovM323);
END_REGION

REGION Network 50: Упоры поштучной выдачи перед зоной оценки
   RUNG wire#powerrail
      I_Contact( "EvaluationZoneThrowOFF_DB".CommonAlarmEvaluationZone )
      Contact( #Run323_timer.Q )
      Contact( "FC_323_1_delayed" )
      wire#w1
      Coil( "HS".Upor_Sorting.OffCom )
      Coil( "UporDispenser_down" )
   END_RUNG
   RUNG wire#w1
      Not()
      Coil( "HS".Upor_Sorting.OnCom )
   END_RUNG
   // the same network as SCL:
   "HS".Upor_Sorting.OffCom := NOT "EvaluationZoneThrowOFF_DB".CommonAlarmEvaluationZone AND #Run323_timer.Q AND "FC_323_1_delayed";
   "UporDispenser_down" := "HS".Upor_Sorting.OffCom;
   "HS".Upor_Sorting.OnCom := NOT "HS".Upor_Sorting.OffCom;
END_REGION

REGION Network 51: M 323 авто вперед (цепь перед поштучкой)
   RUNG wire#powerrail
      I_Contact( "ALG".Alarm_Sorting )
      Contact( "ALG".Auto_Sorting )
      Contact( #HaveSxema )
      wire#w1
      Contact( "M323_RunTask" )
      wire#w2
      Coil( "IM".M_323_Small_Chain.OnCom )
   END_RUNG
   RUNG wire#w1
      Contact( "M323_HoldRun" )
   END_RUNG wire#w2
   // the same network as SCL:
   "IM".M_323_Small_Chain.OnCom := NOT "ALG".Alarm_Sorting AND "ALG".Auto_Sorting AND #HaveSxema AND ("M323_RunTask" OR "M323_HoldRun");
END_REGION

REGION Network 52: Старт ПЧТ M 323
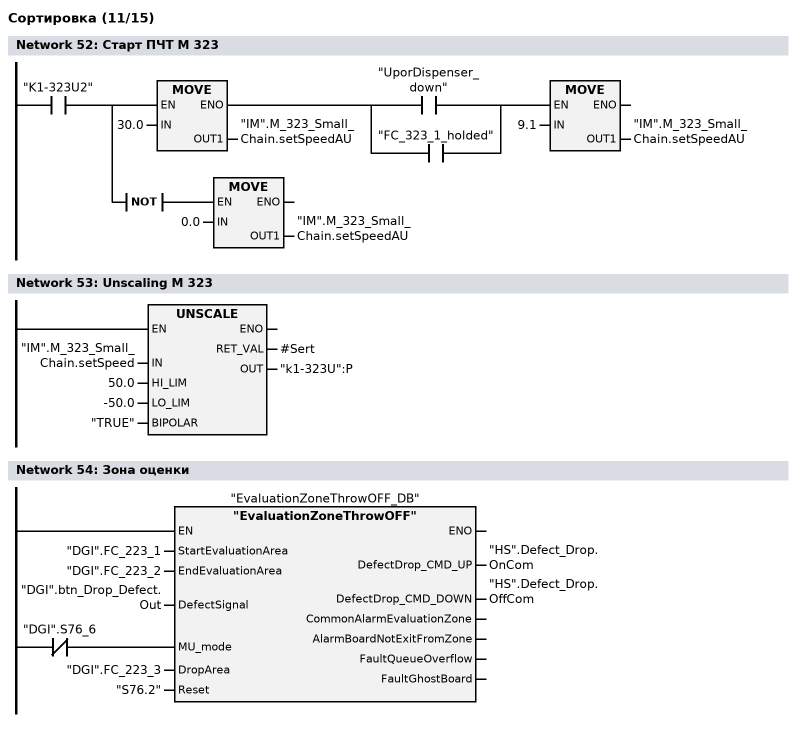
   RUNG wire#powerrail
      Contact( "K1-323U2" )
      wire#w1
      { S7_GenerateENO := "TRUE" } Move(in := 30.0, out1 => "IM".M_323_Small_Chain.setSpeedAU)
      wire#w2
      Contact( "UporDispenser_down" )
      wire#w3
      { S7_GenerateENO := "TRUE" } Move(in := 9.1, out1 => "IM".M_323_Small_Chain.setSpeedAU)
   END_RUNG
   RUNG wire#w2
      Contact( "FC_323_1_holded" )
   END_RUNG wire#w3
   RUNG wire#w1
      Not()
      { S7_GenerateENO := "TRUE" } Move(in := 0.0, out1 => "IM".M_323_Small_Chain.setSpeedAU)
   END_RUNG
   // the same network as SCL:
   // ENO of a box is taken as its EN; it also drops when the box reports an error
   IF "K1-323U2" THEN "IM".M_323_Small_Chain.setSpeedAU := 30.0; END_IF;
   IF "K1-323U2" AND ("UporDispenser_down" OR "FC_323_1_holded") THEN
       "IM".M_323_Small_Chain.setSpeedAU := 9.1;
   END_IF;
   IF NOT "K1-323U2" THEN "IM".M_323_Small_Chain.setSpeedAU := 0.0; END_IF;
END_REGION

REGION Network 53: Unscaling M 323
   RUNG wire#powerrail
      UNSCALE(IN := "IM".M_323_Small_Chain.setSpeed, HI_LIM := 50.0, LO_LIM := -50.0, BIPOLAR := "TRUE", RET_VAL => #Sert, OUT => "k1-323U":P)
   END_RUNG
   // the same network as SCL:
   #Sert := UNSCALE(IN := "IM".M_323_Small_Chain.setSpeed,
                    HI_LIM := 50.0,
                    LO_LIM := -50.0,
                    BIPOLAR := "TRUE",
                    OUT => "k1-323U":P);
END_REGION

REGION Network 54: Зона оценки
   RUNG wire#powerrail
      "EvaluationZoneThrowOFF_DB"(MU_mode := wire#w1, StartEvaluationArea := "DGI".FC_223_1, EndEvaluationArea := "DGI".FC_223_2, DefectSignal := "DGI".btn_Drop_Defect.Out, DropArea := "DGI".FC_223_3, Reset := "S76.2", DefectDrop_CMD_UP => "HS".Defect_Drop.OnCom, DefectDrop_CMD_DOWN => "HS".Defect_Drop.OffCom, CommonAlarmEvaluationZone =>, AlarmBoardNotExitFromZone =>, FaultQueueOverflow =>, FaultGhostBoard =>)
   END_RUNG
   RUNG wire#powerrail
      I_Contact( "DGI".S76_6 )
   END_RUNG wire#w1
   // the same network as SCL:
   "EvaluationZoneThrowOFF_DB"(StartEvaluationArea := "DGI".FC_223_1,   // "EvaluationZoneThrowOFF"
                           EndEvaluationArea := "DGI".FC_223_2,
                           DefectSignal := "DGI".btn_Drop_Defect.Out,
                           MU_mode := NOT "DGI".S76_6,
                           DropArea := "DGI".FC_223_3,
                           Reset := "S76.2",
                           DefectDrop_CMD_UP => "HS".Defect_Drop.OnCom,
                           DefectDrop_CMD_DOWN => "HS".Defect_Drop.OffCom);
END_REGION

REGION Network 55: Измерение длины досок + залипание линейки + управление очередью бобышек под линейкой
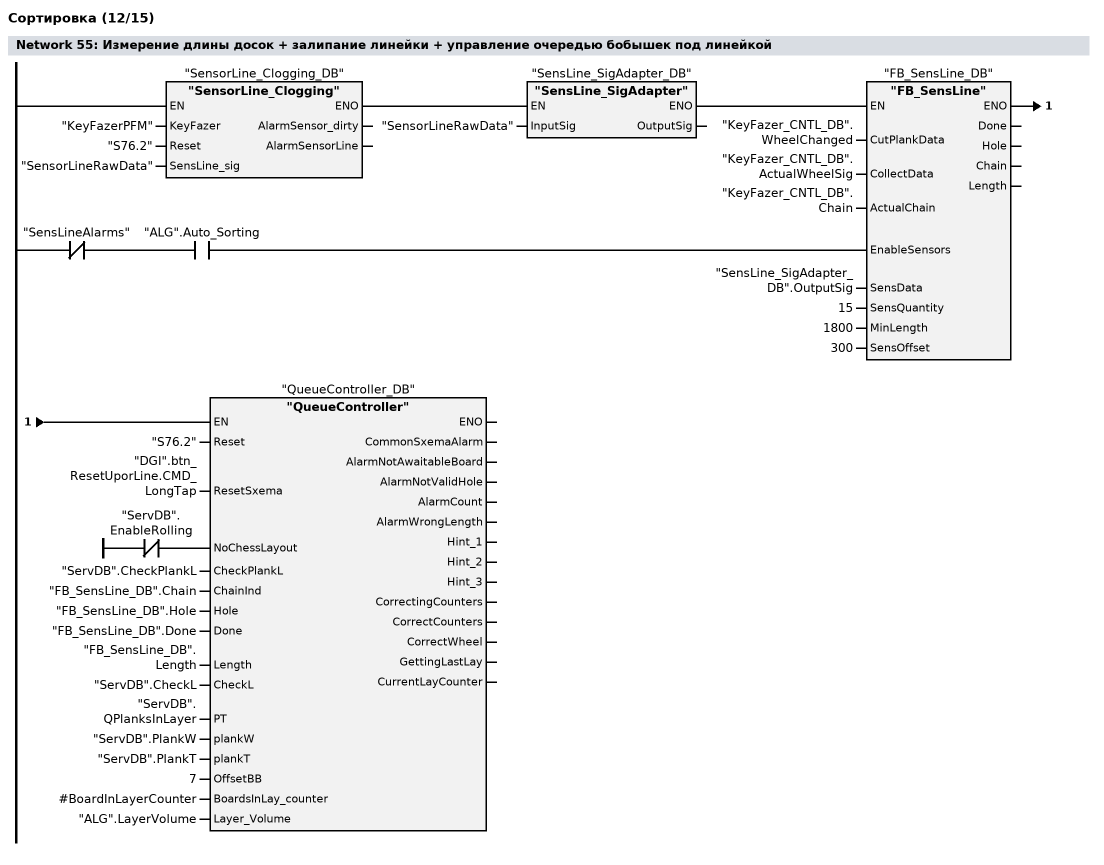
   RUNG wire#powerrail
      "SensorLine_Clogging_DB"(KeyFazer := "KeyFazerPFM", Reset := "S76.2", SensLine_sig := "SensorLineRawData", AlarmSensor_dirty =>, AlarmSensorLine =>)
      "SensLine_SigAdapter_DB"(InputSig := "SensorLineRawData", OutputSig =>)
      "FB_SensLine_DB"(EnableSensors := wire#w1, CutPlankData := "KeyFazer_CNTL_DB".WheelChanged, CollectData := "KeyFazer_CNTL_DB".ActualWheelSig, ActualChain := "KeyFazer_CNTL_DB".Chain, SensData := "SensLine_SigAdapter_DB".OutputSig, SensQuantity := 15, MinLength := 1800, SensOffset := 300, Done =>, Hole =>, Chain =>, Length =>)
      "QueueController_DB"(NoChessLayout := wire#w2, Reset := "S76.2", ResetSxema := "DGI".btn_ResetUporLine.CMD_LongTap, CheckPlankL := "ServDB".CheckPlankL, ChainInd := "FB_SensLine_DB".Chain, Hole := "FB_SensLine_DB".Hole, Done := "FB_SensLine_DB".Done, Length := "FB_SensLine_DB".Length, CheckL := "ServDB".CheckL, PT := "ServDB".QPlanksInLayer, plankW := "ServDB".PlankW, plankT := "ServDB".PlankT, OffsetBB := 7, BoardsInLay_counter := #BoardInLayerCounter, Layer_Volume := "ALG".LayerVolume, CommonSxemaAlarm =>, AlarmNotAwaitableBoard =>, AlarmNotValidHole =>, AlarmCount =>, AlarmWrongLength =>, Hint_1 =>, Hint_2 =>, Hint_3 =>, CorrectingCounters =>, CorrectCounters =>, CorrectWheel =>, GettingLastLay =>, CurrentLayCounter =>)
   END_RUNG
   RUNG wire#powerrail
      I_Contact( "SensLineAlarms" )
      Contact( "ALG".Auto_Sorting )
   END_RUNG wire#w1
   RUNG wire#powerrail
      I_Contact( "ServDB".EnableRolling )
   END_RUNG wire#w2
   // the same network as SCL:
   "SensorLine_Clogging_DB"(KeyFazer := "KeyFazerPFM",   // "SensorLine_Clogging"
                           Reset := "S76.2",
                           SensLine_sig := "SensorLineRawData",
                           ENO => #_w1);
   "SensLine_SigAdapter_DB"(EN := #_w1, InputSig := "SensorLineRawData", ENO => #_w2);   // "SensLine_SigAdapter"
   "FB_SensLine_DB"(EN := #_w2,   // "FB_SensLine"
                    CutPlankData := "KeyFazer_CNTL_DB".WheelChanged,
                    CollectData := "KeyFazer_CNTL_DB".ActualWheelSig,
                    ActualChain := "KeyFazer_CNTL_DB".Chain,
                    EnableSensors := NOT "SensLineAlarms" AND "ALG".Auto_Sorting,
                    SensData := "SensLine_SigAdapter_DB".OutputSig,
                    SensQuantity := 15,
                    MinLength := 1800,
                    SensOffset := 300,
                    ENO => #_w3);
   IF #_w3 THEN
       "QueueController_DB"(Reset := "S76.2",   // "QueueController"
                            ResetSxema := "DGI".btn_ResetUporLine.CMD_LongTap,
                            NoChessLayout := NOT "ServDB".EnableRolling,
                            CheckPlankL := "ServDB".CheckPlankL,
                            ChainInd := "FB_SensLine_DB".Chain,
                            Hole := "FB_SensLine_DB".Hole,
                            Done := "FB_SensLine_DB".Done,
                            Length := "FB_SensLine_DB".Length,
                            CheckL := "ServDB".CheckL,
                            PT := "ServDB".QPlanksInLayer,
                            plankW := "ServDB".PlankW,
                            plankT := "ServDB".PlankT,
                            OffsetBB := 7,
                            BoardsInLay_counter := #BoardInLayerCounter,
                            Layer_Volume := "ALG".LayerVolume);
   END_IF;
END_REGION

REGION Network 56: Управление упорами перед транспортером с бобышками
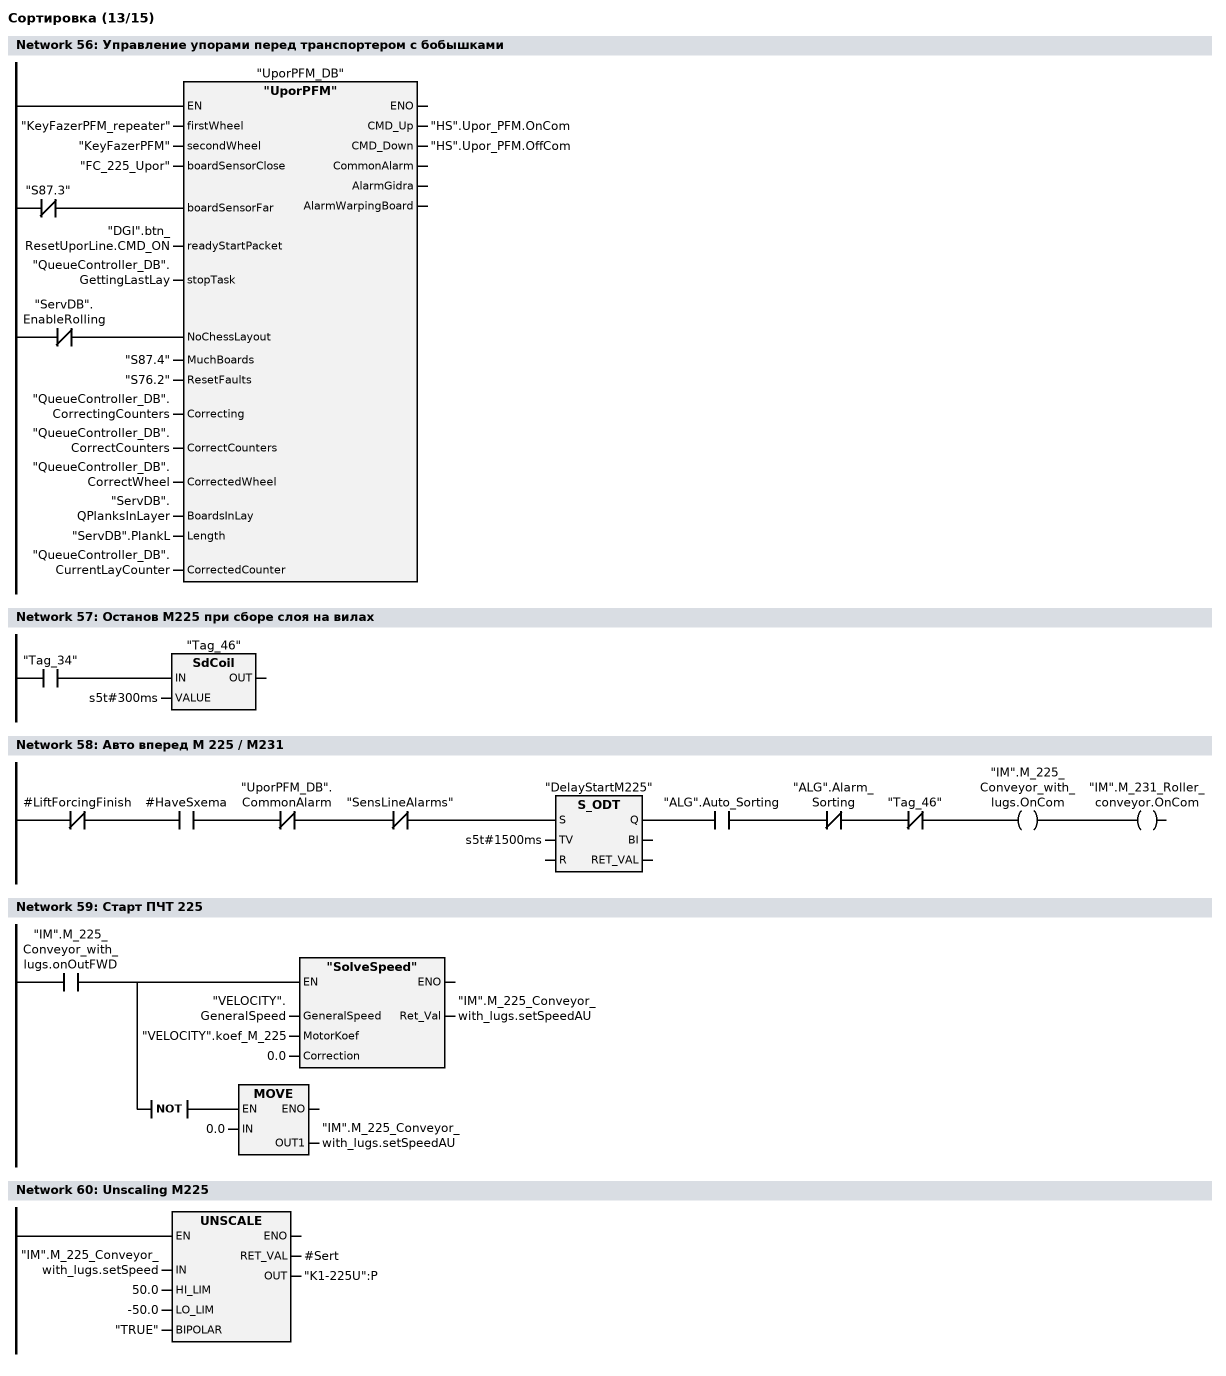
   RUNG wire#powerrail
      "UporPFM_DB"(boardSensorFar := wire#w1, NoChessLayout := wire#w2, firstWheel := "KeyFazerPFM_repeater", secondWheel := "KeyFazerPFM", boardSensorClose := "FC_225_Upor", readyStartPacket := "DGI".btn_ResetUporLine.CMD_ON, stopTask := "QueueController_DB".GettingLastLay, MuchBoards := "S87.4", ResetFaults := "S76.2", Correcting := "QueueController_DB".CorrectingCounters, CorrectCounters := "QueueController_DB".CorrectCounters, CorrectedWheel := "QueueController_DB".CorrectWheel, BoardsInLay := "ServDB".QPlanksInLayer, Length := "ServDB".PlankL, CorrectedCounter := "QueueController_DB".CurrentLayCounter, CMD_Up => "HS".Upor_PFM.OnCom, CMD_Down => "HS".Upor_PFM.OffCom, CommonAlarm =>, AlarmGidra =>, AlarmWarpingBoard =>)
   END_RUNG
   RUNG wire#powerrail
      I_Contact( "S87.3" )
   END_RUNG wire#w1
   RUNG wire#powerrail
      I_Contact( "ServDB".EnableRolling )
   END_RUNG wire#w2
   // the same network as SCL:
   "UporPFM_DB"(firstWheel := "KeyFazerPFM_repeater",   // "UporPFM"
                secondWheel := "KeyFazerPFM",
                boardSensorClose := "FC_225_Upor",
                boardSensorFar := NOT "S87.3",
                readyStartPacket := "DGI".btn_ResetUporLine.CMD_ON,
                stopTask := "QueueController_DB".GettingLastLay,
                NoChessLayout := NOT "ServDB".EnableRolling,
                MuchBoards := "S87.4",
                ResetFaults := "S76.2",
                Correcting := "QueueController_DB".CorrectingCounters,
                CorrectCounters := "QueueController_DB".CorrectCounters,
                CorrectedWheel := "QueueController_DB".CorrectWheel,
                BoardsInLay := "ServDB".QPlanksInLayer,
                Length := "ServDB".PlankL,
                CorrectedCounter := "QueueController_DB".CurrentLayCounter,
                CMD_Up => "HS".Upor_PFM.OnCom,
                CMD_Down => "HS".Upor_PFM.OffCom);
END_REGION

REGION Network 57: Останов M225 при сборе слоя на вилах
   // no SCL statement known for SdCoil: written as a call
   SdCoil(in := "Tag_34", value := s5t#300ms, operand := "Tag_46");
END_REGION

REGION Network 58: Авто вперед M 225 / M231
   RUNG wire#powerrail
      I_Contact( #LiftForcingFinish )
      Contact( #HaveSxema )
      I_Contact( "UporPFM_DB".CommonAlarm )
      I_Contact( "SensLineAlarms" )
      S_ODT(T_NO := "DelayStartM225", TV := s5t#1500ms, R :=, BI =>, RET_VAL =>)
      Contact( "ALG".Auto_Sorting )
      I_Contact( "ALG".Alarm_Sorting )
      I_Contact( "Tag_46" )
      Coil( "IM".M_225_Conveyor_with_lugs.OnCom )
      Coil( "IM".M_231_Roller_conveyor.OnCom )
   END_RUNG
   // the same network as SCL:
   #_s5time1 := S_ODT(T_NO := "DelayStartM225",
                      S := NOT #LiftForcingFinish AND #HaveSxema AND NOT "UporPFM_DB".CommonAlarm AND NOT "SensLineAlarms",
                      TV := s5t#1500ms,
                      Q => #_w1);
   "IM".M_225_Conveyor_with_lugs.OnCom := #_w1 AND "ALG".Auto_Sorting AND NOT "ALG".Alarm_Sorting AND NOT "Tag_46";
   "IM".M_231_Roller_conveyor.OnCom := "IM".M_225_Conveyor_with_lugs.OnCom;
END_REGION

REGION Network 59: Старт ПЧТ 225
   RUNG wire#powerrail
      Contact( "IM".M_225_Conveyor_with_lugs.onOutFWD )
      wire#w1
      "SolveSpeed"(GeneralSpeed := "VELOCITY".GeneralSpeed, MotorKoef := "VELOCITY".koef_M_225, Correction := 0.0, Ret_Val => "IM".M_225_Conveyor_with_lugs.setSpeedAU)
   END_RUNG
   RUNG wire#w1
      Not()
      { S7_GenerateENO := "TRUE" } Move(in := 0.0, out1 => "IM".M_225_Conveyor_with_lugs.setSpeedAU)
   END_RUNG
   // the same network as SCL:
   #_w1 := "IM".M_225_Conveyor_with_lugs.onOutFWD;
   IF #_w1 THEN
       "IM".M_225_Conveyor_with_lugs.setSpeedAU := "SolveSpeed"(GeneralSpeed := "VELOCITY".GeneralSpeed,
                               MotorKoef := "VELOCITY".koef_M_225,
                               Correction := 0.0);
   END_IF;
   IF NOT #_w1 THEN "IM".M_225_Conveyor_with_lugs.setSpeedAU := 0.0; END_IF;
END_REGION

REGION Network 60: Unscaling M225
   RUNG wire#powerrail
      UNSCALE(IN := "IM".M_225_Conveyor_with_lugs.setSpeed, HI_LIM := 50.0, LO_LIM := -50.0, BIPOLAR := "TRUE", RET_VAL => #Sert, OUT => "K1-225U":P)
   END_RUNG
   // the same network as SCL:
   #Sert := UNSCALE(IN := "IM".M_225_Conveyor_with_lugs.setSpeed,
                    HI_LIM := 50.0,
                    LO_LIM := -50.0,
                    BIPOLAR := "TRUE",
                    OUT => "K1-225U":P);
END_REGION

REGION Network 61: Старт ПЧТ 231
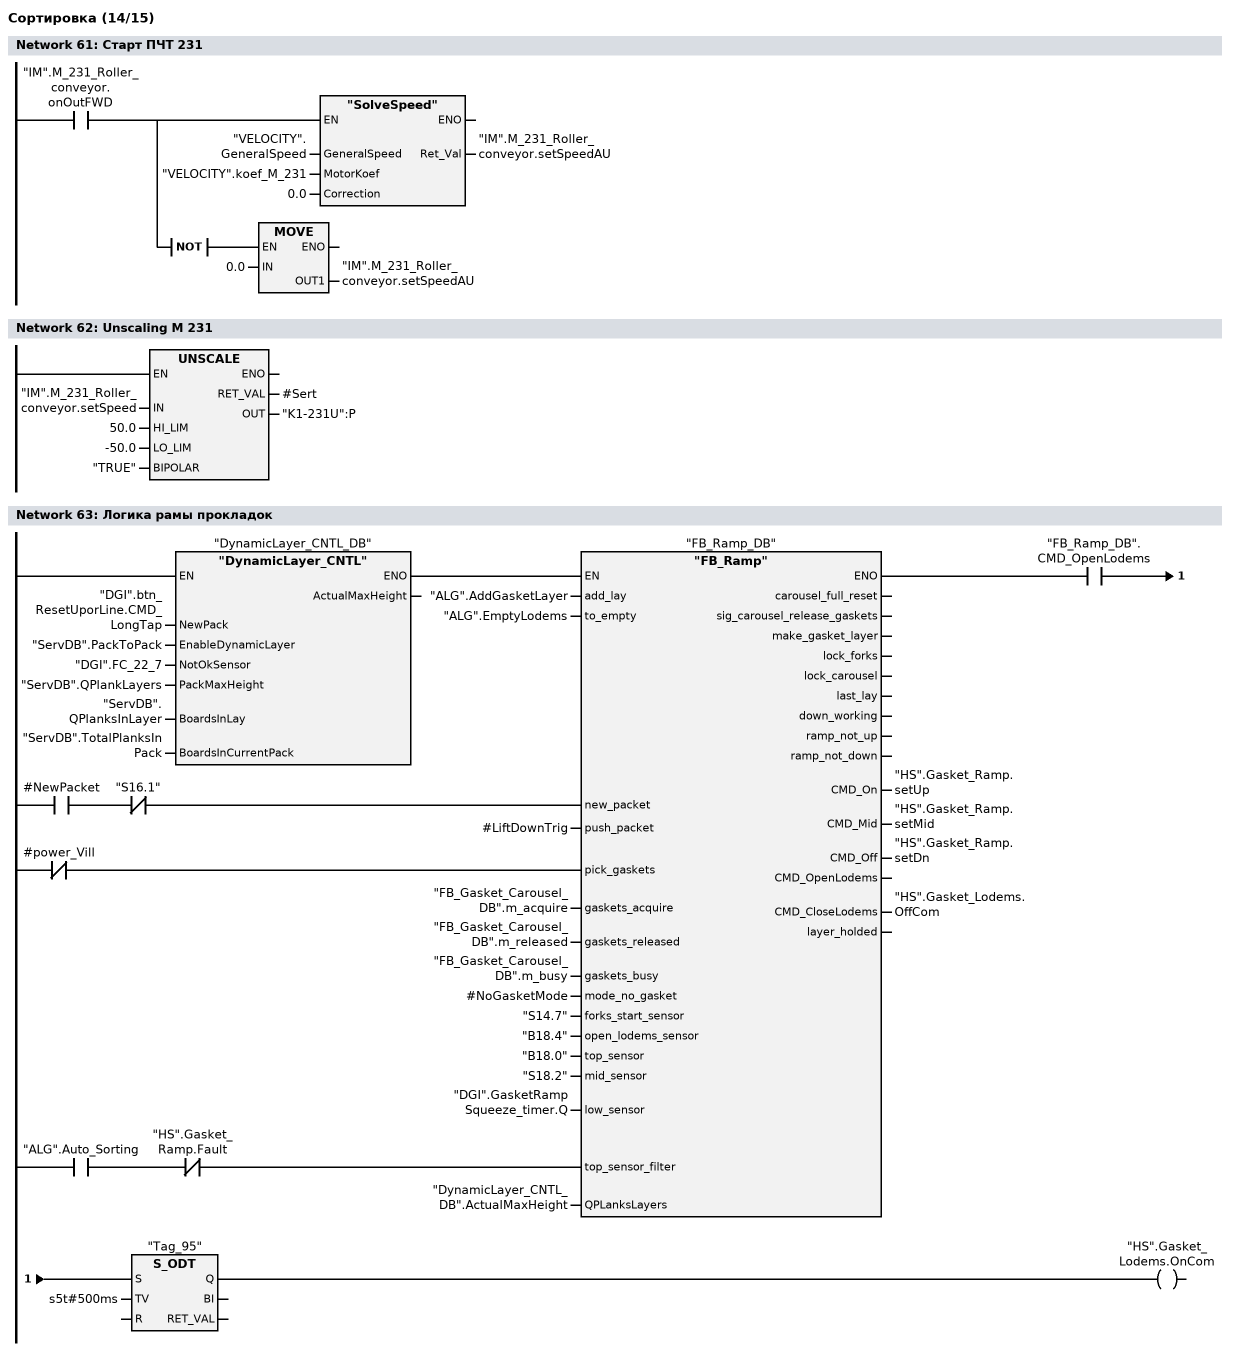
   RUNG wire#powerrail
      Contact( "IM".M_231_Roller_conveyor.onOutFWD )
      wire#w1
      "SolveSpeed"(GeneralSpeed := "VELOCITY".GeneralSpeed, MotorKoef := "VELOCITY".koef_M_231, Correction := 0.0, Ret_Val => "IM".M_231_Roller_conveyor.setSpeedAU)
   END_RUNG
   RUNG wire#w1
      Not()
      { S7_GenerateENO := "TRUE" } Move(in := 0.0, out1 => "IM".M_231_Roller_conveyor.setSpeedAU)
   END_RUNG
   // the same network as SCL:
   #_w1 := "IM".M_231_Roller_conveyor.onOutFWD;
   IF #_w1 THEN
       "IM".M_231_Roller_conveyor.setSpeedAU := "SolveSpeed"(GeneralSpeed := "VELOCITY".GeneralSpeed,
                               MotorKoef := "VELOCITY".koef_M_231,
                               Correction := 0.0);
   END_IF;
   IF NOT #_w1 THEN "IM".M_231_Roller_conveyor.setSpeedAU := 0.0; END_IF;
END_REGION

REGION Network 62: Unscaling M 231
   RUNG wire#powerrail
      UNSCALE(IN := "IM".M_231_Roller_conveyor.setSpeed, HI_LIM := 50.0, LO_LIM := -50.0, BIPOLAR := "TRUE", RET_VAL => #Sert, OUT => "K1-231U":P)
   END_RUNG
   // the same network as SCL:
   #Sert := UNSCALE(IN := "IM".M_231_Roller_conveyor.setSpeed,
                    HI_LIM := 50.0,
                    LO_LIM := -50.0,
                    BIPOLAR := "TRUE",
                    OUT => "K1-231U":P);
END_REGION

REGION Network 63: Логика рамы прокладок
   RUNG wire#powerrail
      "DynamicLayer_CNTL_DB"(NewPack := "DGI".btn_ResetUporLine.CMD_LongTap, EnableDynamicLayer := "ServDB".PackToPack, NotOkSensor := "DGI".FC_22_7, PackMaxHeight := "ServDB".QPlankLayers, BoardsInLay := "ServDB".QPlanksInLayer, BoardsInCurrentPack := "ServDB".TotalPlanksInPack, ActualMaxHeight =>)
      "FB_Ramp_DB"(new_packet := wire#w1, pick_gaskets := wire#w2, top_sensor_filter := wire#w3, add_lay := "ALG".AddGasketLayer, to_empty := "ALG".EmptyLodems, push_packet := #LiftDownTrig, gaskets_acquire := "FB_Gasket_Carousel_DB".m_acquire, gaskets_released := "FB_Gasket_Carousel_DB".m_released, gaskets_busy := "FB_Gasket_Carousel_DB".m_busy, mode_no_gasket := #NoGasketMode, forks_start_sensor := "S14.7", open_lodems_sensor := "B18.4", top_sensor := "B18.0", mid_sensor := "S18.2", low_sensor := "DGI".GasketRampSqueeze_timer.Q, QPLanksLayers := "DynamicLayer_CNTL_DB".ActualMaxHeight, carousel_full_reset =>, sig_carousel_release_gaskets =>, make_gasket_layer =>, lock_forks =>, lock_carousel =>, last_lay =>, down_working =>, ramp_not_up =>, ramp_not_down =>, CMD_On => "HS".Gasket_Ramp.setUp, CMD_Mid => "HS".Gasket_Ramp.setMid, CMD_Off => "HS".Gasket_Ramp.setDn, CMD_OpenLodems =>, CMD_CloseLodems => "HS".Gasket_Lodems.OffCom, layer_holded =>)
      Contact( "FB_Ramp_DB".CMD_OpenLodems )
      S_ODT(T_NO := "Tag_95", TV := s5t#500ms, R :=, BI =>, RET_VAL =>)
      Coil( "HS".Gasket_Lodems.OnCom )
   END_RUNG
   RUNG wire#powerrail
      Contact( #NewPacket )
      I_Contact( "S16.1" )
   END_RUNG wire#w1
   RUNG wire#powerrail
      I_Contact( #power_Vill )
   END_RUNG wire#w2
   RUNG wire#powerrail
      Contact( "ALG".Auto_Sorting )
      I_Contact( "HS".Gasket_Ramp.Fault )
   END_RUNG wire#w3
   // the same network as SCL:
   "DynamicLayer_CNTL_DB"(NewPack := "DGI".btn_ResetUporLine.CMD_LongTap,   // "DynamicLayer_CNTL"
                          EnableDynamicLayer := "ServDB".PackToPack,
                          NotOkSensor := "DGI".FC_22_7,
                          PackMaxHeight := "ServDB".QPlankLayers,
                          BoardsInLay := "ServDB".QPlanksInLayer,
                          BoardsInCurrentPack := "ServDB".TotalPlanksInPack,
                          ENO => #_w1);
   "FB_Ramp_DB"(EN := #_w1,   // "FB_Ramp"
                add_lay := "ALG".AddGasketLayer,
                to_empty := "ALG".EmptyLodems,
                new_packet := #NewPacket AND NOT "S16.1",
                push_packet := #LiftDownTrig,
                pick_gaskets := NOT #power_Vill,
                gaskets_acquire := "FB_Gasket_Carousel_DB".m_acquire,
                gaskets_released := "FB_Gasket_Carousel_DB".m_released,
                gaskets_busy := "FB_Gasket_Carousel_DB".m_busy,
                mode_no_gasket := #NoGasketMode,
                forks_start_sensor := "S14.7",
                open_lodems_sensor := "B18.4",
                top_sensor := "B18.0",
                mid_sensor := "S18.2",
                low_sensor := "DGI".GasketRampSqueeze_timer.Q,
                top_sensor_filter := "ALG".Auto_Sorting AND NOT "HS".Gasket_Ramp.Fault,
                QPLanksLayers := "DynamicLayer_CNTL_DB".ActualMaxHeight,
                CMD_On => "HS".Gasket_Ramp.setUp,
                CMD_Mid => "HS".Gasket_Ramp.setMid,
                CMD_Off => "HS".Gasket_Ramp.setDn,
                CMD_CloseLodems => "HS".Gasket_Lodems.OffCom,
                ENO => #_w2);
   #_s5time1 := S_ODT(T_NO := "Tag_95", S := #_w2 AND "FB_Ramp_DB".CMD_OpenLodems, TV := s5t#500ms, Q => #_w3);
   "HS".Gasket_Lodems.OnCom := #_w3;
END_REGION

REGION Network 64: Новый пакет
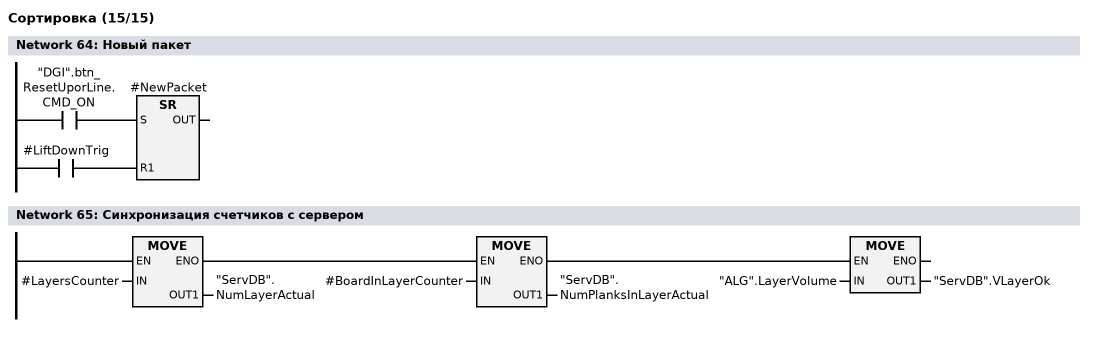
   RUNG wire#powerrail
      Contact( "DGI".btn_ResetUporLine.CMD_ON )
      S_SR(operand := #NewPacket, r1 := wire#w1)
   END_RUNG
   RUNG wire#powerrail
      Contact( #LiftDownTrig )
   END_RUNG wire#w1
   // the same network as SCL:
   IF "DGI".btn_ResetUporLine.CMD_ON THEN
       #NewPacket := TRUE;   // SR flip-flop
   END_IF;
   IF #LiftDownTrig THEN #NewPacket := FALSE; END_IF;
END_REGION

REGION Network 65: Синхронизация счетчиков с сервером
   RUNG wire#powerrail
      { S7_GenerateENO := "TRUE" } Move(in := #LayersCounter, out1 => "ServDB".NumLayerActual)
      { S7_GenerateENO := "TRUE" } Move(in := #BoardInLayerCounter, out1 => "ServDB".NumPlanksInLayerActual)
      { S7_GenerateENO := "TRUE" } Move(in := "ALG".LayerVolume, out1 => "ServDB".VLayerOk)
   END_RUNG
   // the same network as SCL:
   // ENO of a box is taken as its EN; it also drops when the box reports an error
   "ServDB".NumLayerActual := #LayersCounter;
   "ServDB".NumPlanksInLayerActual := #BoardInLayerCounter;
   "ServDB".VLayerOk := "ALG".LayerVolume;
END_REGION
END_FUNCTION_BLOCK
